C03628=1135.696,-18.528,-48.394,179.412,6.258,149.306
C03629=1135.690,-18.279,-48.406,179.415,6.260,149.305
C03630=1135.685,-18.029,-48.419,179.417,6.261,149.305
C03631=1135.680,-17.780,-48.431,179.420,6.261,149.304
C03632=1135.675,-17.530,-48.443,179.422,6.262,149.304
C03633=1135.669,-17.280,-48.455,179.424,6.263,149.303
C03634=1135.664,-17.031,-48.468,179.427,6.263,149.303
C03635=1135.659,-16.781,-48.480,179.429,6.264,149.302
C03636=1135.654,-16.532,-48.492,179.431,6.265,149.302
C03637=1135.649,-16.282,-48.505,179.434,6.265,149.301
C03638=1135.643,-16.032,-48.517,179.437,6.267,149.300
C03639=1135.639,-15.782,-48.530,179.439,6.267,149.300
C03640=1135.633,-15.533,-48.542,179.442,6.268,149.299
C03641=1135.628,-15.283,-48.554,179.444,6.269,149.299
C03642=1135.623,-15.034,-48.567,179.446,6.269,149.298
C03643=1135.617,-14.784,-48.579,179.449,6.270,149.298
C03644=1135.612,-14.534,-48.592,179.451,6.271,149.297
C03645=1135.607,-14.285,-48.605,179.453,6.271,149.297
C03646=1135.601,-14.036,-48.617,179.456,6.273,149.296
C03647=1135.597,-13.785,-48.629,179.458,6.273,149.296
C03648=1135.591,-13.536,-48.642,179.461,6.274,149.295
C03649=1135.586,-13.286,-48.655,179.463,6.275,149.294
C03650=1135.581,-13.036,-48.667,179.465,6.275,149.294
C03651=1135.576,-12.787,-48.679,179.468,6.276,149.293
C03652=1135.571,-12.538,-48.692,179.470,6.277,149.293
C03653=1135.566,-12.288,-48.705,179.473,6.278,149.292
C03654=1135.561,-12.038,-48.717,179.476,6.279,149.292
C03655=1135.555,-11.788,-48.730,179.478,6.279,149.291
C03656=1135.550,-11.539,-48.742,179.480,6.280,149.291
C03657=1135.545,-11.290,-48.755,179.483,6.281,149.290
C03658=1135.540,-11.039,-48.767,179.485,6.281,149.290
C03659=1135.535,-10.790,-48.780,179.487,6.282,149.289
C03660=1135.529,-10.540,-48.792,179.490,6.283,149.288
C03661=1135.524,-10.291,-48.805,179.493,6.284,149.288
C03662=1135.519,-10.042,-48.818,179.495,6.285,149.287
C03663=1135.514,-9.791,-48.830,179.497,6.285,149.287
C03664=1135.509,-9.541,-48.843,179.500,6.286,149.286
C03665=1135.503,-9.292,-48.856,179.502,6.287,149.286
C03666=1135.498,-9.043,-48.868,179.505,6.288,149.285
C03667=1135.494,-8.793,-48.881,179.507,6.289,149.285
C03668=1135.488,-8.543,-48.894,179.509,6.290,149.284
C03669=1135.483,-8.294,-48.907,179.512,6.290,149.283
C03670=1135.478,-8.045,-48.920,179.514,6.291,149.283
C03671=1135.473,-7.794,-48.932,179.516,6.292,149.283
C03672=1135.468,-7.545,-48.944,179.520,6.293,149.282
C03673=1135.462,-7.295,-48.958,179.522,6.294,149.281
C03674=1135.457,-7.046,-48.970,179.524,6.295,149.281
C03675=1135.452,-6.796,-48.983,179.527,6.295,149.280
C03676=1135.447,-6.546,-48.996,179.529,6.296,149.280
C03677=1135.441,-6.297,-49.009,179.532,6.297,149.279
C03678=1135.436,-6.047,-49.022,179.534,6.298,149.279
C03679=1135.432,-5.797,-49.035,179.536,6.299,149.278
C03680=1135.426,-5.548,-49.047,179.539,6.299,149.277
C03681=1135.421,-5.298,-49.060,179.541,6.300,149.277
C03682=1135.415,-5.049,-49.073,179.544,6.301,149.276
C03683=1135.411,-4.799,-49.086,179.547,6.302,149.276
C03684=1135.405,-4.549,-49.099,179.549,6.303,149.275
C03685=1135.400,-4.300,-49.112,179.551,6.303,149.275
C03686=1135.395,-4.050,-49.125,179.554,6.304,149.274
C03687=1135.390,-3.801,-49.137,179.557,6.305,149.274
C03688=1135.384,-3.551,-49.151,179.559,6.306,149.273
C03689=1135.380,-3.301,-49.163,179.561,6.307,149.273
C03690=1135.375,-3.052,-49.176,179.564,6.307,149.272
C03691=1135.369,-2.802,-49.189,179.566,6.308,149.272
C03692=1135.364,-2.552,-49.202,179.569,6.309,149.271
C03693=1135.359,-2.303,-49.215,179.571,6.310,149.270
C03694=1135.353,-2.053,-49.228,179.573,6.311,149.270
C03695=1135.349,-1.803,-49.241,179.576,6.311,149.269
C03696=1135.343,-1.554,-49.255,179.578,6.312,149.269
C03697=1135.338,-1.305,-49.268,179.581,6.314,149.268
C03698=1135.334,-1.055,-49.280,179.584,6.314,149.268
C03699=1135.328,-0.805,-49.294,179.586,6.315,149.267
C03700=1135.323,-0.556,-49.306,179.588,6.316,149.267
C03701=1135.317,-0.306,-49.320,179.591,6.317,149.266
C03702=1135.312,-0.056,-49.332,179.593,6.318,149.266
C03703=1135.308,0.192,-49.346,179.596,6.319,149.265
C03704=1135.302,0.443,-49.359,179.598,6.319,149.264
C03705=1135.297,0.692,-49.372,179.600,6.320,149.264
C03706=1135.291,0.962,-49.386,179.604,6.321,149.263
C03707=1135.287,1.231,-49.401,179.606,6.322,149.263
C03708=1135.280,1.501,-49.415,179.609,6.323,149.262
C03709=1135.275,1.771,-49.429,179.611,6.324,149.262
C03710=1135.270,2.019,-49.442,179.614,6.324,149.261
C03711=1135.265,2.270,-49.456,179.617,6.326,149.261
C03712=1135.259,2.519,-49.468,179.619,6.327,149.260
C03713=1135.254,2.769,-49.482,179.622,6.327,149.259
C03714=1135.249,3.018,-49.495,179.624,6.328,149.259
C03715=1135.243,3.268,-49.508,179.626,6.330,149.258
C03716=1135.239,3.518,-49.521,179.629,6.330,149.258
C03717=1135.233,3.767,-49.535,179.631,6.331,149.257
C03718=1135.229,4.017,-49.548,179.633,6.332,149.257
C03719=1135.223,4.266,-49.561,179.637,6.333,149.256
C03720=1135.219,4.516,-49.574,179.639,6.334,149.256
C03721=1135.213,4.765,-49.588,179.641,6.334,149.255
C03722=1135.208,5.015,-49.601,179.644,6.335,149.255
C03723=1135.203,5.265,-49.614,179.647,6.336,149.254
C03724=1135.198,5.514,-49.628,179.649,6.337,149.253
C03725=1135.192,5.764,-49.641,179.651,6.338,149.253
C03726=1135.188,6.013,-49.655,179.654,6.339,149.252
C03727=1135.182,6.263,-49.668,179.657,6.340,149.252
C03728=1135.177,6.512,-49.681,179.659,6.341,149.251
C03729=1135.172,6.762,-49.695,179.661,6.341,149.251
C03730=1135.166,7.012,-49.708,179.664,6.342,149.250
C03731=1135.162,7.261,-49.722,179.667,6.343,149.250
C03732=1135.156,7.511,-49.735,179.669,6.344,149.249
C03733=1135.152,7.761,-49.748,179.671,6.345,149.249
C03734=1135.146,8.010,-49.762,179.674,6.346,149.248
C03735=1135.141,8.260,-49.776,179.676,6.347,149.248
C03736=1135.136,8.509,-49.789,179.679,6.347,149.247
C03737=1135.131,8.759,-49.802,179.681,6.348,149.246
C03738=1135.125,9.008,-49.816,179.684,6.350,149.246
C03739=1135.121,9.258,-49.829,179.687,6.350,149.245
C03740=1135.116,9.508,-49.844,179.689,6.351,149.245
C03741=1135.111,9.757,-49.856,179.692,6.353,149.244
C03742=1135.106,10.007,-49.870,179.694,6.353,149.244
C03743=1135.100,10.256,-49.884,179.696,6.354,149.243
C03744=1135.096,10.506,-49.897,179.699,6.356,149.243
C03745=1135.090,10.756,-49.911,179.702,6.356,149.242
C03746=1135.085,11.005,-49.925,179.704,6.357,149.242
C03747=1135.080,11.255,-49.937,179.706,6.358,149.241
C03748=1135.075,11.504,-49.952,179.709,6.359,149.240
C03749=1135.069,11.753,-49.966,179.712,6.360,149.240
C03750=1135.064,12.004,-49.979,179.714,6.360,149.240
C03751=1135.060,12.253,-49.993,179.717,6.362,149.239
C03752=1135.054,12.503,-50.006,179.719,6.362,149.238
C03753=1135.049,12.752,-50.020,179.722,6.363,149.238
C03754=1135.044,13.001,-50.034,179.725,6.364,149.237
C03755=1135.039,13.251,-50.047,179.727,6.365,149.237
C03756=1135.034,13.501,-50.061,179.729,6.366,149.236
C03757=1135.028,13.750,-50.075,179.732,6.367,149.236
C03758=1135.024,14.000,-50.088,179.734,6.368,149.235
C03759=1135.018,14.249,-50.102,179.737,6.369,149.235
C03760=1135.013,14.499,-50.117,179.740,6.370,149.234
C03761=1135.008,14.749,-50.130,179.742,6.371,149.234
C03762=1135.003,14.998,-50.144,179.745,6.371,149.233
C03763=1134.998,15.248,-50.158,179.747,6.373,149.232
C03764=1134.993,15.497,-50.171,179.750,6.374,149.232
C03765=1134.988,15.747,-50.185,179.752,6.374,149.231
C03766=1134.983,15.997,-50.199,179.755,6.376,149.231
C03767=1134.977,16.246,-50.213,179.757,6.377,149.230
C03768=1134.973,16.496,-50.226,179.760,6.377,149.230
C03769=1134.968,16.745,-50.241,179.763,6.379,149.229
C03770=1134.962,16.994,-50.255,179.765,6.380,149.229
C03771=1134.957,17.244,-50.269,179.767,6.380,149.228
C03772=1134.952,17.494,-50.282,179.770,6.382,149.228
C03773=1134.946,17.743,-50.296,179.772,6.382,149.227
C03774=1134.942,17.993,-50.310,179.775,6.383,149.226
C03775=1134.937,18.243,-50.324,179.778,6.384,149.226
C03776=1134.932,18.492,-50.338,179.780,6.385,149.226
C03777=1134.926,18.742,-50.352,179.783,6.386,149.225
C03778=1134.921,18.992,-50.366,179.785,6.387,149.224
C03779=1134.916,19.241,-50.380,179.788,6.388,149.224
C03780=1134.911,19.490,-50.394,179.790,6.389,149.223
C03781=1134.906,19.740,-50.408,179.793,6.390,149.223
C03782=1134.902,19.989,-50.422,179.795,6.391,149.222
C03783=1134.896,20.238,-50.436,179.798,6.391,149.222
C03784=1134.891,20.488,-50.450,179.801,6.393,149.221
C03785=1134.886,20.738,-50.464,179.803,6.394,149.221
C03786=1134.880,20.987,-50.478,179.806,6.395,149.220
C03787=1134.875,21.237,-50.492,179.808,6.396,149.220
C03788=1134.870,21.487,-50.506,179.810,6.397,149.219
C03789=1134.865,21.737,-50.521,179.814,6.398,149.219
C03790=1134.860,21.986,-50.535,179.816,6.399,149.218
C03791=1134.855,22.235,-50.549,179.818,6.400,149.218
C03792=1134.850,22.485,-50.563,179.821,6.401,149.217
C03793=1134.845,22.735,-50.577,179.823,6.402,149.216
C03794=1134.839,22.984,-50.591,179.826,6.403,149.216
C03795=1134.834,23.233,-50.606,179.829,6.404,149.215
C03796=1134.830,23.483,-50.620,179.831,6.404,149.215
C03797=1134.825,23.733,-50.634,179.834,6.406,149.214
C03798=1134.819,23.982,-50.648,179.836,6.407,149.214
C03799=1134.814,24.232,-50.662,179.839,6.408,149.213
C03800=1134.809,24.481,-50.677,179.841,6.409,149.213
C03801=1134.804,24.731,-50.691,179.844,6.409,149.212
C03802=1134.799,24.981,-50.705,179.847,6.411,149.212
C03803=1134.794,25.230,-50.719,179.849,6.412,149.211
C03804=1134.789,25.479,-50.733,179.852,6.413,149.211
C03805=1134.784,25.729,-50.748,179.854,6.414,149.210
C03806=1134.779,25.978,-50.763,179.856,6.415,149.210
C03807=1134.774,26.228,-50.777,179.860,6.416,149.209
C03808=1134.769,26.477,-50.791,179.862,6.417,149.208
C03809=1134.764,26.727,-50.805,179.865,6.418,149.208
C03810=1134.757,26.996,-50.821,179.867,6.419,149.207
C03811=1134.752,27.265,-50.836,179.870,6.420,149.207
C03812=1134.747,27.534,-50.852,179.873,6.421,149.206
C03813=1134.742,27.803,-50.867,179.876,6.422,149.206
C03814=1134.737,28.053,-50.881,179.878,6.423,149.205
C03815=1134.731,28.302,-50.897,179.881,6.425,149.205
C03816=1134.726,28.552,-50.911,179.884,6.425,149.204
C03817=1134.721,28.801,-50.925,179.886,6.427,149.204
C03818=1134.716,29.051,-50.939,179.888,6.427,149.203
C03819=1134.711,29.301,-50.954,179.891,6.429,149.203
C03820=1134.706,29.550,-50.969,179.894,6.429,149.202
C03821=1134.701,29.799,-50.983,179.896,6.430,149.201
C03822=1134.696,30.049,-50.998,179.899,6.432,149.201
C03823=1134.690,30.298,-51.012,179.901,6.432,149.200
C03824=1134.686,30.548,-51.027,179.904,6.434,149.200
C03825=1134.681,30.797,-51.041,179.906,6.435,149.199
C03826=1134.676,31.047,-51.055,179.910,6.436,149.199
C03827=1134.671,31.296,-51.070,179.912,6.437,149.198
C03828=1134.665,31.546,-51.085,179.915,6.439,149.198
C03829=1134.660,31.796,-51.099,179.917,6.439,149.197
C03830=1134.656,32.045,-51.114,179.919,6.440,149.197
C03831=1134.651,32.295,-51.129,179.922,6.441,149.196
C03832=1134.645,32.545,-51.144,179.925,6.442,149.196
C03833=1134.640,32.794,-51.159,179.928,6.443,149.195
C03834=1134.635,33.043,-51.173,179.930,6.444,149.195
C03835=1134.630,33.292,-51.187,179.933,6.446,149.194
C03836=1134.624,33.542,-51.202,179.935,6.446,149.194
C03837=1134.620,33.792,-51.217,179.938,6.448,149.193
C03838=1134.615,34.041,-51.231,179.941,6.448,149.192
C03839=1134.610,34.290,-51.246,179.943,6.450,149.192
C03840=1134.604,34.540,-51.261,179.946,6.451,149.192
C03841=1134.600,34.789,-51.276,179.948,6.451,149.191
C03842=1134.595,35.039,-51.290,179.951,6.453,149.190
C03843=1134.589,35.289,-51.306,179.953,6.454,149.190
C03844=1134.584,35.538,-51.320,179.956,6.455,149.189
C03845=1134.579,35.788,-51.334,179.959,6.456,149.189
C03846=1134.574,36.037,-51.350,179.961,6.457,149.188
C03847=1134.569,36.287,-51.364,179.964,6.458,149.188
C03848=1134.564,36.536,-51.379,179.967,6.460,149.187
C03849=1134.559,36.786,-51.394,179.969,6.460,149.187
C03850=1134.554,37.035,-51.409,179.972,6.462,149.186
C03851=1134.549,37.285,-51.423,179.974,6.462,149.186
C03852=1134.544,37.534,-51.439,179.977,6.464,149.185
C03853=1134.539,37.784,-51.454,179.979,6.465,149.185
C03854=1134.533,38.034,-51.469,179.982,6.466,149.184
C03855=1134.529,38.283,-51.484,179.985,6.467,149.184
C03856=1134.524,38.532,-51.498,179.987,6.469,149.183
C03857=1134.518,38.782,-51.513,179.990,6.469,149.183
C03858=1134.513,39.031,-51.528,179.993,6.471,149.182
C03859=1134.508,39.281,-51.543,179.995,6.471,149.182
C03860=1134.503,39.530,-51.558,179.998,6.473,149.181
C03861=1134.498,39.780,-51.573,-180.000,6.474,149.180
C03862=1134.493,40.029,-51.588,-179.997,6.475,149.180
C03863=1134.488,40.279,-51.602,-179.994,6.476,149.179
C03864=1134.483,40.528,-51.618,-179.991,6.477,149.179
C03865=1134.479,40.778,-51.633,-179.989,6.478,149.178
C03866=1134.473,41.028,-51.648,-179.987,6.480,149.178
C03867=1134.468,41.277,-51.663,-179.984,6.480,149.177
C03868=1134.463,41.526,-51.679,-179.981,6.482,149.177
C03869=1134.458,41.776,-51.693,-179.979,6.483,149.176
C03870=1134.453,42.026,-51.709,-179.976,6.484,149.176
C03871=1134.448,42.275,-51.724,-179.974,6.485,149.175
C03872=1134.442,42.524,-51.739,-179.971,6.486,149.175
C03873=1134.438,42.774,-51.754,-179.968,6.487,149.174
C03874=1134.432,43.023,-51.769,-179.965,6.488,149.174
C03875=1134.428,43.273,-51.785,-179.963,6.489,149.173
C03876=1134.423,43.522,-51.800,-179.960,6.490,149.173
C03877=1134.418,43.772,-51.814,-179.957,6.492,149.172
C03878=1134.412,44.022,-51.830,-179.955,6.493,149.172
C03879=1134.408,44.271,-51.845,-179.952,6.495,149.171
C03880=1134.402,44.520,-51.861,-179.950,6.495,149.171
C03881=1134.398,44.769,-51.876,-179.947,6.497,149.170
C03882=1134.392,45.019,-51.890,-179.945,6.497,149.170
C03883=1134.388,45.269,-51.906,-179.942,6.499,149.169
C03884=1134.383,45.518,-51.921,-179.939,6.500,149.169
C03885=1134.377,45.768,-51.937,-179.937,6.501,149.168
C03886=1134.373,46.017,-51.952,-179.934,6.502,149.167
C03887=1134.367,46.266,-51.968,-179.931,6.503,149.167
C03888=1134.362,46.516,-51.982,-179.928,6.505,149.167
C03889=1134.357,46.766,-51.998,-179.926,6.506,149.166
C03890=1134.352,47.015,-52.013,-179.923,6.507,149.165
C03891=1134.347,47.265,-52.028,-179.921,6.508,149.165
C03892=1134.342,47.514,-52.044,-179.918,6.509,149.165
C03893=1134.337,47.763,-52.060,-179.915,6.510,149.164
C03894=1134.333,48.013,-52.075,-179.913,6.512,149.163
C03895=1134.327,48.263,-52.090,-179.911,6.512,149.163
C03896=1134.322,48.512,-52.105,-179.908,6.514,149.163
C03897=1134.317,48.761,-52.121,-179.905,6.515,149.162
C03898=1134.312,49.010,-52.137,-179.902,6.516,149.161
C03899=1134.308,49.260,-52.152,-179.900,6.518,149.161
C03900=1134.302,49.510,-52.168,-179.897,6.518,149.160
C03901=1134.297,49.759,-52.183,-179.894,6.520,149.160
C03902=1134.292,50.008,-52.199,-179.892,6.521,149.159
C03903=1134.287,50.258,-52.214,-179.889,6.522,149.159
C03904=1134.282,50.508,-52.230,-179.886,6.524,149.158
C03905=1134.277,50.757,-52.245,-179.884,6.524,149.158
C03906=1134.272,51.006,-52.260,-179.881,6.526,149.157
C03907=1134.267,51.256,-52.276,-179.878,6.526,149.157
C03908=1134.262,51.506,-52.292,-179.876,6.528,149.156
C03909=1134.256,51.755,-52.307,-179.873,6.530,149.156
C03910=1134.252,52.005,-52.323,-179.871,6.531,149.155
C03911=1134.247,52.254,-52.338,-179.868,6.532,149.155
C03912=1134.242,52.504,-52.354,-179.865,6.533,149.154
C03913=1134.237,52.752,-52.370,-179.863,6.534,149.154
C03914=1134.231,53.021,-52.387,-179.859,6.536,149.153
C03915=1134.226,53.290,-52.403,-179.857,6.537,149.153
C03916=1134.221,53.559,-52.420,-179.854,6.538,149.152
C03917=1134.215,53.827,-52.437,-179.851,6.539,149.152
C03918=1134.210,54.077,-52.453,-179.848,6.541,149.151
C03919=1134.205,54.327,-52.469,-179.846,6.541,149.151
C03920=1134.200,54.576,-52.485,-179.843,6.543,149.150
C03921=1134.195,54.825,-52.500,-179.840,6.545,149.150
C03922=1134.191,55.075,-52.516,-179.838,6.545,149.149
C03923=1134.185,55.324,-52.532,-179.835,6.547,149.149
C03924=1134.180,55.574,-52.547,-179.833,6.548,149.148
C03925=1134.175,55.823,-52.564,-179.830,6.549,149.148
C03926=1134.170,56.073,-52.580,-179.827,6.550,149.147
C03927=1134.165,56.322,-52.595,-179.825,6.551,149.147
C03928=1134.160,56.572,-52.611,-179.822,6.553,149.146
C03929=1134.156,56.820,-52.627,-179.819,6.555,149.146
C03930=1134.150,57.070,-52.642,-179.816,6.555,149.145
C03931=1134.145,57.320,-52.658,-179.814,6.557,149.145
C03932=1134.140,57.569,-52.675,-179.812,6.557,149.144
C03933=1134.135,57.818,-52.690,-179.808,6.559,149.143
C03934=1134.130,58.068,-52.706,-179.806,6.560,149.143
C03935=1134.125,58.317,-52.723,-179.803,6.561,149.143
C03936=1134.120,58.567,-52.738,-179.801,6.563,149.142
C03937=1134.115,58.817,-52.754,-179.797,6.564,149.142
C03938=1134.110,59.065,-52.770,-179.795,6.565,149.141
C03939=1134.105,59.315,-52.786,-179.793,6.567,149.141
C03940=1134.100,59.564,-52.803,-179.790,6.568,149.140
C03941=1134.095,59.814,-52.819,-179.787,6.569,149.140
C03942=1134.090,60.064,-52.834,-179.784,6.570,149.139
C03943=1134.085,60.313,-52.850,-179.782,6.572,149.139
C03944=1134.080,60.563,-52.866,-179.779,6.573,149.138
C03945=1134.075,60.811,-52.883,-179.776,6.574,149.138
C03946=1134.070,61.062,-52.899,-179.773,6.576,149.137
C03947=1134.065,61.310,-52.915,-179.771,6.577,149.137
C03948=1134.060,61.560,-52.931,-179.769,6.578,149.136
C03949=1134.055,61.809,-52.947,-179.765,6.579,149.136
C03950=1134.050,62.059,-52.963,-179.763,6.580,149.135
C03951=1134.045,62.308,-52.980,-179.760,6.582,149.135
C03952=1134.040,62.558,-52.995,-179.757,6.583,149.134
C03953=1134.035,62.807,-53.012,-179.755,6.584,149.134
C03954=1134.030,63.056,-53.027,-179.752,6.586,149.133
C03955=1134.025,63.306,-53.044,-179.749,6.587,149.133
C03956=1134.020,63.555,-53.060,-179.747,6.588,149.132
C03957=1134.016,63.805,-53.076,-179.744,6.589,149.132
C03958=1134.010,64.054,-53.092,-179.741,6.591,149.131
C03959=1134.006,64.304,-53.109,-179.739,6.592,149.131
C03960=1134.001,64.552,-53.125,-179.736,6.593,149.130
C03961=1133.995,64.803,-53.141,-179.733,6.595,149.130
C03962=1133.991,65.052,-53.158,-179.731,6.596,149.129
C03963=1133.985,65.302,-53.174,-179.728,6.597,149.129
C03964=1133.981,65.551,-53.190,-179.725,6.599,149.128
C03965=1133.976,65.800,-53.207,-179.723,6.599,149.128
C03966=1133.971,66.050,-53.223,-179.720,6.601,149.127
C03967=1133.966,66.299,-53.239,-179.717,6.603,149.127
C03968=1133.961,66.548,-53.256,-179.715,6.604,149.126
C03969=1133.955,66.798,-53.272,-179.712,6.605,149.126
C03970=1133.951,67.048,-53.288,-179.709,6.607,149.125
C03971=1133.946,67.296,-53.305,-179.707,6.608,149.125
C03972=1133.941,67.546,-53.321,-179.704,6.609,149.124
C03973=1133.936,67.796,-53.337,-179.701,6.610,149.124
C03974=1133.931,68.045,-53.354,-179.698,6.612,149.123
C03975=1133.926,68.294,-53.371,-179.696,6.614,149.123
C03976=1133.921,68.544,-53.386,-179.693,6.614,149.122
C03977=1133.916,68.793,-53.403,-179.690,6.616,149.122
C03978=1133.911,69.042,-53.419,-179.687,6.617,149.121
C03979=1133.906,69.292,-53.437,-179.685,6.618,149.121
C03980=1133.901,69.541,-53.453,-179.683,6.620,149.120
C03981=1133.896,69.791,-53.469,-179.679,6.621,149.120
C03982=1133.892,70.040,-53.486,-179.677,6.623,149.119
C03983=1133.886,70.289,-53.503,-179.674,6.624,149.119
C03984=1133.881,70.539,-53.519,-179.672,6.625,149.118
C03985=1133.877,70.788,-53.536,-179.669,6.627,149.118
C03986=1133.871,71.037,-53.553,-179.666,6.628,149.117
C03987=1133.866,71.288,-53.569,-179.664,6.629,149.117
C03988=1133.862,71.537,-53.585,-179.661,6.631,149.117
C03989=1133.857,71.786,-53.602,-179.658,6.632,149.116
C03990=1133.851,72.036,-53.619,-179.655,6.633,149.115
C03991=1133.846,72.284,-53.635,-179.653,6.634,149.115
C03992=1133.842,72.534,-53.652,-179.650,6.636,149.115
C03993=1133.837,72.784,-53.669,-179.647,6.638,149.114
C03994=1133.832,73.032,-53.686,-179.645,6.639,149.114
C03995=1133.827,73.282,-53.702,-179.642,6.640,149.113
C03996=1133.822,73.532,-53.719,-179.639,6.641,149.113
C03997=1133.817,73.781,-53.736,-179.636,6.643,149.112
C03998=1133.812,74.030,-53.753,-179.634,6.645,149.112
C03999=1133.807,74.280,-53.770,-179.631,6.645,149.111
C04000=1133.803,74.529,-53.786,-179.628,6.647,149.111
C04001=1133.797,74.778,-53.803,-179.625,6.649,149.110
C04002=1133.792,75.028,-53.820,-179.623,6.650,149.110
C04003=1133.787,75.278,-53.837,-179.621,6.651,149.109
C04004=1133.782,75.526,-53.853,-179.617,6.652,149.109
C04005=1133.778,75.776,-53.870,-179.615,6.654,149.108
C04006=1133.772,76.026,-53.887,-179.612,6.656,149.108
C04007=1133.768,76.275,-53.904,-179.610,6.656,149.107
C04008=1133.762,76.524,-53.921,-179.607,6.658,149.107
C04009=1133.758,76.774,-53.938,-179.604,6.659,149.106
C04010=1133.752,77.024,-53.955,-179.601,6.661,149.106
C04011=1133.747,77.272,-53.971,-179.598,6.663,149.105
C04012=1133.742,77.522,-53.989,-179.596,6.664,149.105
C04013=1133.738,77.771,-54.006,-179.593,6.665,149.105
C04014=1133.733,78.021,-54.023,-179.590,6.667,149.104
C04015=1133.728,78.270,-54.039,-179.587,6.668,149.104
C04016=1133.722,78.519,-54.057,-179.585,6.669,149.103
C04017=1133.718,78.769,-54.073,-179.582,6.671,149.103
C04018=1133.712,79.038,-54.092,-179.579,6.672,149.102
C04019=1133.707,79.306,-54.110,-179.576,6.674,149.102
C04020=1133.702,79.575,-54.129,-179.574,6.675,149.101
C04021=1133.697,79.842,-54.147,-179.570,6.677,149.101
C04022=1133.692,80.092,-54.164,-179.568,6.678,149.100
C04023=1133.686,80.341,-54.181,-179.565,6.680,149.100
C04024=1133.682,80.591,-54.198,-179.562,6.681,149.099
C04025=1133.677,80.840,-54.216,-179.559,6.683,149.099
C04026=1133.672,81.089,-54.232,-179.557,6.684,149.098
C04027=1133.667,81.339,-54.250,-179.554,6.685,149.098
C04028=1133.662,81.588,-54.266,-179.551,6.687,149.097
C04029=1133.657,81.837,-54.284,-179.549,6.689,149.097
C04030=1133.652,82.087,-54.302,-179.546,6.690,149.096
C04031=1133.648,82.337,-54.318,-179.543,6.691,149.096
C04032=1133.642,82.585,-54.336,-179.540,6.692,149.095
C04033=1133.637,82.835,-54.353,-179.538,6.694,149.095
C04034=1133.632,83.084,-54.370,-179.535,6.696,149.095
C04035=1133.628,83.333,-54.388,-179.532,6.697,149.094
C04036=1133.623,83.583,-54.404,-179.529,6.699,149.093
C04037=1133.618,83.832,-54.422,-179.527,6.699,149.093
C04038=1133.613,84.082,-54.440,-179.524,6.701,149.093
C04039=1133.608,84.331,-54.456,-179.521,6.703,149.092
C04040=1133.603,84.580,-54.474,-179.519,6.704,149.092
C04041=1133.598,84.830,-54.491,-179.516,6.706,149.091
C04042=1133.594,85.079,-54.509,-179.513,6.707,149.091
C04043=1133.588,85.328,-54.526,-179.510,6.708,149.090
C04044=1133.583,85.577,-54.544,-179.508,6.710,149.090
C04045=1133.578,85.827,-54.561,-179.505,6.712,149.089
C04046=1133.574,86.076,-54.579,-179.502,6.713,149.089
C04047=1133.569,86.326,-54.596,-179.500,6.715,149.089
C04048=1133.564,86.575,-54.614,-179.496,6.716,149.088
C04049=1133.559,86.825,-54.631,-179.494,6.718,149.087
C04050=1133.554,87.073,-54.648,-179.491,6.719,149.087
C04051=1133.549,87.323,-54.665,-179.489,6.720,149.087
C04052=1133.544,87.572,-54.683,-179.486,6.722,149.086
C04053=1133.539,87.822,-54.701,-179.483,6.724,149.086
C04054=1133.534,88.071,-54.718,-179.480,6.725,149.085
C04055=1133.529,88.320,-54.736,-179.477,6.727,149.085
C04056=1133.524,88.570,-54.753,-179.474,6.728,149.084
C04057=1133.519,88.819,-54.771,-179.472,6.730,149.084
C04058=1133.514,89.069,-54.788,-179.470,6.731,149.083
C04059=1133.510,89.318,-54.806,-179.467,6.732,149.083
C04060=1133.505,89.567,-54.824,-179.464,6.734,149.082
C04061=1133.500,89.816,-54.841,-179.461,6.735,149.082
C04062=1133.495,90.066,-54.859,-179.458,6.737,149.082
C04063=1133.490,90.315,-54.877,-179.455,6.739,149.081
C04064=1133.485,90.565,-54.894,-179.453,6.740,149.081
C04065=1133.481,90.813,-54.912,-179.450,6.742,149.080
C04066=1133.476,91.063,-54.930,-179.448,6.743,149.080
C04067=1133.470,91.312,-54.947,-179.445,6.744,149.079
C04068=1133.466,91.562,-54.965,-179.442,6.746,149.079
C04069=1133.461,91.811,-54.983,-179.439,6.748,149.078
C04070=1133.456,92.060,-55.001,-179.436,6.749,149.078
C04071=1133.450,92.310,-55.018,-179.434,6.751,149.077
C04072=1133.446,92.559,-55.036,-179.431,6.753,149.077
C04073=1133.441,92.808,-55.054,-179.428,6.754,149.077
C04074=1133.436,93.057,-55.071,-179.425,6.755,149.076
C04075=1133.431,93.307,-55.089,-179.422,6.757,149.076
C04076=1133.426,93.556,-55.107,-179.420,6.758,149.075
C04077=1133.421,93.805,-55.125,-179.417,6.760,149.075
C04078=1133.417,94.054,-55.143,-179.414,6.761,149.074
C04079=1133.412,94.304,-55.161,-179.412,6.763,149.074
C04080=1133.407,94.553,-55.179,-179.409,6.765,149.073
C04081=1133.402,94.803,-55.196,-179.406,6.766,149.073
C04082=1133.397,95.052,-55.214,-179.403,6.768,149.072
C04083=1133.392,95.302,-55.232,-179.400,6.769,149.072
C04084=1133.387,95.551,-55.250,-179.398,6.771,149.072
C04085=1133.382,95.800,-55.268,-179.395,6.773,149.071
C04086=1133.378,96.049,-55.286,-179.392,6.774,149.071
C04087=1133.373,96.298,-55.304,-179.389,6.776,149.070
C04088=1133.368,96.547,-55.322,-179.387,6.778,149.070
C04089=1133.363,96.797,-55.340,-179.384,6.778,149.069
C04090=1133.358,97.046,-55.358,-179.381,6.780,149.069
C04091=1133.354,97.296,-55.376,-179.378,6.781,149.068
C04092=1133.349,97.545,-55.394,-179.376,6.783,149.068
C04093=1133.343,97.794,-55.413,-179.373,6.785,149.068
C04094=1133.338,98.043,-55.431,-179.370,6.786,149.067
C04095=1133.333,98.293,-55.449,-179.368,6.788,149.067
C04096=1133.328,98.542,-55.467,-179.365,6.790,149.066
C04097=1133.324,98.792,-55.485,-179.362,6.791,149.066
C04098=1133.319,99.041,-55.503,-179.359,6.793,149.065
C04099=1133.314,99.290,-55.521,-179.356,6.794,149.065
C04100=1133.309,99.539,-55.539,-179.353,6.796,149.064
C04101=1133.304,99.788,-55.557,-179.351,6.798,149.064
C04102=1133.300,100.038,-55.576,-179.348,6.799,149.064
C04103=1133.294,100.288,-55.594,-179.345,6.801,149.063
C04104=1133.289,100.537,-55.612,-179.342,6.803,149.063
C04105=1133.285,100.786,-55.630,-179.340,6.804,149.062
C04106=1133.280,101.035,-55.649,-179.337,6.806,149.062
C04107=1133.276,101.285,-55.667,-179.334,6.808,149.062
C04108=1133.271,101.534,-55.685,-179.331,6.809,149.061
C04109=1133.265,101.783,-55.704,-179.328,6.811,149.060
C04110=1133.260,102.032,-55.722,-179.325,6.812,149.060
C04111=1133.255,102.282,-55.740,-179.323,6.814,149.060
C04112=1133.251,102.531,-55.759,-179.320,6.816,149.059
C04113=1133.246,102.780,-55.777,-179.318,6.817,149.059
C04114=1133.241,103.029,-55.795,-179.315,6.818,149.058
C04115=1133.236,103.279,-55.813,-179.312,6.820,149.058
C04116=1133.232,103.528,-55.832,-179.310,6.822,149.058
C04117=1133.227,103.777,-55.850,-179.307,6.823,149.057
C04118=1133.221,104.027,-55.869,-179.304,6.825,149.057
C04119=1133.216,104.276,-55.887,-179.301,6.826,149.056
C04120=1133.212,104.525,-55.906,-179.298,6.828,149.056
C04121=1133.207,104.774,-55.924,-179.295,6.830,149.055
C04122=1133.202,105.043,-55.944,-179.292,6.832,149.055
C04123=1133.196,105.311,-55.963,-179.289,6.834,149.054
C04124=1133.191,105.579,-55.984,-179.287,6.835,149.054
C04125=1133.186,105.848,-56.004,-179.283,6.837,149.053
C04126=1133.181,106.097,-56.022,-179.281,6.838,149.053
C04127=1133.176,106.346,-56.041,-179.278,6.840,149.053
C04128=1133.172,106.596,-56.059,-179.275,6.842,149.052
C04129=1133.166,106.845,-56.078,-179.273,6.843,149.052
C04130=1133.162,107.094,-56.097,-179.270,6.845,149.051
C04131=1133.157,107.344,-56.115,-179.267,6.847,149.051
C04132=1133.152,107.593,-56.134,-179.264,6.848,149.051
C04133=1133.147,107.842,-56.152,-179.262,6.850,149.050
C04134=1133.143,108.092,-56.171,-179.259,6.852,149.050
C04135=1133.137,108.341,-56.190,-179.256,6.853,149.049
C04136=1133.133,108.590,-56.208,-179.253,6.856,149.049
C04137=1133.128,108.839,-56.228,-179.250,6.858,149.048
C04138=1133.123,109.088,-56.246,-179.247,6.859,149.048
C04139=1133.118,109.337,-56.264,-179.244,6.861,149.047
C04140=1133.113,109.587,-56.283,-179.241,6.862,149.047
C04141=1133.109,109.836,-56.302,-179.239,6.864,149.047
C04142=1133.104,110.086,-56.321,-179.236,6.866,149.046
C04143=1133.099,110.334,-56.339,-179.233,6.867,149.046
C04144=1133.094,110.583,-56.359,-179.230,6.869,149.045
C04145=1133.089,110.833,-56.377,-179.228,6.871,149.045
C04146=1133.084,111.082,-56.396,-179.225,6.872,149.045
C04147=1133.079,111.331,-56.414,-179.222,6.874,149.044
C04148=1133.074,111.581,-56.434,-179.219,6.876,149.044
C04149=1133.070,111.829,-56.453,-179.217,6.877,149.043
C04150=1133.065,112.080,-56.472,-179.214,6.879,149.043
C04151=1133.060,112.328,-56.490,-179.211,6.881,149.043
C04152=1133.055,112.578,-56.509,-179.209,6.882,149.042
C04153=1133.050,112.827,-56.528,-179.206,6.884,149.042
C04154=1133.045,113.076,-56.547,-179.203,6.886,149.041
C04155=1133.041,113.326,-56.566,-179.200,6.887,149.041
C04156=1133.035,113.575,-56.585,-179.198,6.889,149.040
C04157=1133.031,113.824,-56.604,-179.194,6.891,149.040
C04158=1133.026,114.073,-56.623,-179.192,6.893,149.040
C04159=1133.021,114.323,-56.642,-179.189,6.895,149.039
C04160=1133.016,114.571,-56.661,-179.186,6.896,149.039
C04161=1133.012,114.821,-56.681,-179.183,6.898,149.038
C04162=1133.007,115.070,-56.699,-179.181,6.900,149.038
C04163=1133.002,115.320,-56.718,-179.178,6.902,149.038
C04164=1132.997,115.569,-56.738,-179.175,6.903,149.037
C04165=1132.993,115.818,-56.757,-179.172,6.905,149.037
C04166=1132.987,116.067,-56.776,-179.169,6.906,149.036
C04167=1132.983,116.317,-56.794,-179.166,6.908,149.036
C04168=1132.978,116.565,-56.814,-179.164,6.910,149.035
C04169=1132.973,116.815,-56.833,-179.160,6.912,149.035
C04170=1132.968,117.064,-56.852,-179.158,6.914,149.035
C04171=1132.964,117.313,-56.872,-179.155,6.915,149.034
C04172=1132.958,117.562,-56.891,-179.152,6.917,149.034
C04173=1132.954,117.811,-56.910,-179.150,6.919,149.033
C04174=1132.949,118.061,-56.928,-179.147,6.920,149.033
C04175=1132.944,118.310,-56.948,-179.144,6.922,149.033
C04176=1132.939,118.559,-56.967,-179.141,6.924,149.032
C04177=1132.934,118.808,-56.986,-179.139,6.925,149.032
C04178=1132.929,119.057,-57.006,-179.136,6.927,149.031
C04179=1132.924,119.307,-57.025,-179.133,6.930,149.031
C04180=1132.920,119.556,-57.044,-179.130,6.931,149.031
C04181=1132.915,119.805,-57.064,-179.127,6.933,149.030
C04182=1132.910,120.055,-57.083,-179.124,6.935,149.030
C04183=1132.905,120.303,-57.103,-179.122,6.936,149.029
C04184=1132.901,120.553,-57.122,-179.119,6.938,149.029
C04185=1132.896,120.802,-57.141,-179.116,6.940,149.029
C04186=1132.891,121.051,-57.161,-179.113,6.941,149.028
C04187=1132.886,121.301,-57.180,-179.110,6.944,149.028
C04188=1132.881,121.549,-57.199,-179.107,6.946,149.027
C04189=1132.877,121.799,-57.219,-179.105,6.947,149.027
C04190=1132.872,122.048,-57.238,-179.102,6.949,149.027
C04191=1132.867,122.297,-57.258,-179.100,6.951,149.026
C04192=1132.862,122.546,-57.278,-179.097,6.953,149.026
C04193=1132.857,122.795,-57.297,-179.094,6.954,149.026
C04194=1132.853,123.044,-57.316,-179.091,6.957,149.025
C04195=1132.848,123.294,-57.336,-179.088,6.959,149.025
C04196=1132.843,123.543,-57.355,-179.085,6.960,149.024
C04197=1132.838,123.792,-57.375,-179.083,6.962,149.024
C04198=1132.833,124.042,-57.395,-179.080,6.964,149.024
C04199=1132.828,124.290,-57.415,-179.077,6.965,149.023
C04200=1132.823,124.540,-57.434,-179.074,6.967,149.023
C04201=1132.819,124.789,-57.453,-179.071,6.969,149.022
C04202=1132.814,125.038,-57.473,-179.068,6.971,149.022
C04203=1132.809,125.287,-57.492,-179.066,6.973,149.022
C04204=1132.805,125.536,-57.513,-179.063,6.974,149.021
C04205=1132.800,125.786,-57.532,-179.060,6.976,149.021
C04206=1132.795,126.035,-57.552,-179.058,6.978,149.020
C04207=1132.790,126.284,-57.571,-179.054,6.980,149.020
C04208=1132.786,126.533,-57.592,-179.051,6.982,149.020
C04209=1132.780,126.782,-57.611,-179.049,6.984,149.019
C04210=1132.776,127.032,-57.631,-179.046,6.985,149.019
C04211=1132.771,127.281,-57.651,-179.043,6.987,149.018
C04212=1132.766,127.530,-57.671,-179.041,6.989,149.018
C04213=1132.761,127.779,-57.690,-179.037,6.991,149.018
C04214=1132.757,128.028,-57.710,-179.035,6.993,149.017
C04215=1132.752,128.278,-57.730,-179.032,6.995,149.017
C04216=1132.747,128.527,-57.750,-179.030,6.997,149.017
C04217=1132.742,128.775,-57.770,-179.027,6.998,149.016
C04218=1132.737,129.025,-57.789,-179.024,7.001,149.016
C04219=1132.733,129.274,-57.810,-179.021,7.003,149.015
C04220=1132.728,129.524,-57.829,-179.018,7.004,149.015
C04221=1132.723,129.772,-57.849,-179.015,7.006,149.015
C04222=1132.718,130.021,-57.869,-179.013,7.008,149.014
C04223=1132.714,130.271,-57.889,-179.009,7.010,149.014
C04224=1132.709,130.520,-57.909,-179.007,7.012,149.013
C04225=1132.705,130.769,-57.929,-179.004,7.013,149.013
C04226=1132.699,131.038,-57.951,-179.001,7.015,149.013
C04227=1132.694,131.306,-57.972,-178.998,7.018,149.012
C04228=1132.688,131.575,-57.993,-178.995,7.019,149.012
C04229=1132.683,131.843,-58.015,-178.992,7.022,149.011
C04230=1132.679,132.092,-58.035,-178.989,7.023,149.011
C04231=1132.674,132.341,-58.055,-178.986,7.025,149.011
C04232=1132.669,132.591,-58.075,-178.984,7.027,149.010
C04233=1132.664,132.840,-58.096,-178.980,7.029,149.010
C04234=1132.660,133.090,-58.116,-178.978,7.031,149.010
C04235=1132.655,133.338,-58.136,-178.975,7.033,149.009
C04236=1132.650,133.587,-58.156,-178.972,7.034,149.009
C04237=1132.645,133.836,-58.176,-178.969,7.037,149.009
C04238=1132.641,134.085,-58.196,-178.967,7.039,149.008
C04239=1132.636,134.335,-58.217,-178.964,7.041,149.008
C04240=1132.631,134.584,-58.237,-178.961,7.042,149.007
C04241=1132.627,134.833,-58.257,-178.958,7.044,149.007
C04242=1132.622,135.082,-58.277,-178.955,7.047,149.007
C04243=1132.616,135.331,-58.297,-178.952,7.048,149.006
C04244=1132.612,135.580,-58.318,-178.950,7.050,149.006
C04245=1132.607,135.829,-58.338,-178.947,7.052,149.005
C04246=1132.602,136.079,-58.358,-178.944,7.054,149.005
C04247=1132.597,136.328,-58.379,-178.941,7.056,149.005
C04248=1132.593,136.577,-58.399,-178.939,7.058,149.004
C04249=1132.588,136.826,-58.419,-178.936,7.060,149.004
C04250=1132.584,137.075,-58.439,-178.933,7.062,149.004
C04251=1132.578,137.325,-58.460,-178.930,7.064,149.003
C04252=1132.574,137.574,-58.480,-178.927,7.065,149.003
C04253=1132.570,137.823,-58.501,-178.924,7.067,149.003
C04254=1132.564,138.072,-58.522,-178.921,7.070,149.002
C04255=1132.560,138.321,-58.542,-178.918,7.071,149.002
C04256=1132.555,138.570,-58.561,-178.916,7.073,149.002
C04257=1132.549,138.819,-58.582,-178.913,7.076,149.001
C04258=1132.530,139.892,-58.674,-179.676,8.531,149.554
C04259=1132.525,140.141,-58.694,-179.675,8.535,149.554
C04260=1132.520,140.391,-58.715,-179.673,8.538,149.554
C04261=1132.516,140.640,-58.736,-179.672,8.541,149.555
C04262=1132.511,140.889,-58.757,-179.670,8.545,149.555
C04263=1132.506,141.138,-58.777,-179.669,8.548,149.555
C04264=1132.501,141.386,-58.799,-179.668,8.551,149.556
C04265=1132.497,141.635,-58.819,-179.666,8.554,149.556
C04266=1132.492,141.885,-58.840,-179.665,8.557,149.557
C04267=1132.488,142.134,-58.861,-179.662,8.561,149.557
C04268=1132.483,142.384,-58.882,-179.661,8.564,149.557
C04269=1132.478,142.633,-58.902,-179.660,8.567,149.558
C04270=1132.473,142.881,-58.924,-179.658,8.571,149.558
C04271=1132.468,143.130,-58.945,-179.657,8.574,149.558
C04272=1132.464,143.379,-58.965,-179.656,8.577,149.559
C04273=1132.459,143.629,-58.986,-179.654,8.580,149.559
C04274=1132.455,143.878,-59.008,-179.653,8.583,149.559
C04275=1132.449,144.159,-59.031,-179.652,8.587,149.560
C04276=1132.444,144.440,-59.055,-179.650,8.591,149.560
C04277=1132.439,144.722,-59.079,-179.648,8.595,149.561
C04278=1132.433,145.004,-59.102,-179.647,8.599,149.561
C04279=1132.428,145.253,-59.124,-179.644,8.603,149.561
C04280=1132.424,145.501,-59.144,-179.641,8.607,149.561
C04281=1132.419,145.751,-59.165,-179.639,8.610,149.562
C04282=1132.414,146.000,-59.187,-179.636,8.615,149.562
C04283=1132.410,146.249,-59.207,-179.633,8.619,149.562
C04284=1132.405,146.498,-59.229,-179.630,8.623,149.562
C04285=1132.400,146.747,-59.250,-179.627,8.627,149.562
C04286=1132.395,146.996,-59.270,-179.624,8.631,149.562
C04287=1132.391,147.245,-59.292,-179.622,8.635,149.563
C04288=1132.386,147.494,-59.313,-179.618,8.639,149.563
C04289=1132.381,147.743,-59.335,-179.616,8.643,149.563
C04290=1132.377,147.992,-59.355,-179.613,8.646,149.563
C04291=1132.372,148.241,-59.378,-179.611,8.651,149.563
C04292=1132.367,148.491,-59.398,-179.607,8.655,149.563
C04293=1132.362,148.739,-59.420,-179.605,8.659,149.563
C04294=1132.358,148.988,-59.441,-179.602,8.663,149.564
C04295=1132.354,149.238,-59.463,-179.599,8.666,149.564
C04296=1132.348,149.487,-59.484,-179.597,8.671,149.564
C04297=1132.344,149.736,-59.505,-179.594,8.674,149.564
C04298=1132.339,149.984,-59.527,-179.591,8.679,149.564
C04299=1132.334,150.234,-59.548,-179.588,8.682,149.564
C04300=1132.330,150.482,-59.569,-179.586,8.686,149.564
C04301=1132.325,150.732,-59.590,-179.582,8.690,149.564
C04302=1132.321,150.981,-59.612,-179.580,8.693,149.564
C04303=1132.316,151.230,-59.634,-179.577,8.697,149.565
C04304=1132.311,151.479,-59.655,-179.574,8.701,149.565
C04305=1132.306,151.728,-59.677,-179.572,8.705,149.565
C04306=1132.301,151.977,-59.699,-179.569,8.709,149.565
C04307=1132.296,152.226,-59.720,-179.566,8.713,149.565
C04308=1132.292,152.476,-59.742,-179.564,8.716,149.565
C04309=1132.287,152.724,-59.763,-179.561,8.720,149.565
C04310=1132.282,152.973,-59.785,-179.558,8.723,149.565
C04311=1132.278,153.222,-59.807,-179.555,8.727,149.565
C04312=1132.273,153.471,-59.828,-179.553,8.731,149.566
C04313=1132.269,153.720,-59.849,-179.550,8.735,149.566
C04314=1132.264,153.969,-59.871,-179.547,8.739,149.566
C04315=1132.259,154.218,-59.893,-179.545,8.742,149.566
C04316=1132.255,154.467,-59.915,-179.542,8.746,149.566
C04317=1132.250,154.716,-59.937,-179.539,8.749,149.566
C04318=1132.245,154.965,-59.959,-179.536,8.753,149.566
C04319=1132.240,155.215,-59.980,-179.534,8.756,149.566
C04320=1132.235,155.463,-60.002,-179.531,8.761,149.567
C04321=1132.231,155.713,-60.024,-179.529,8.764,149.567
C04322=1132.226,155.961,-60.046,-179.526,8.767,149.567
C04323=1132.222,156.211,-60.068,-179.523,8.771,149.567
C04324=1132.217,156.459,-60.089,-179.521,8.774,149.567
C04325=1132.212,156.708,-60.111,-179.518,8.778,149.567
C04326=1132.208,156.957,-60.133,-179.516,8.781,149.567
C04327=1132.204,157.171,-60.152,-179.513,8.785,149.567
C04328=1132.200,157.387,-60.171,-179.511,8.788,149.567
C04329=1132.196,157.601,-60.190,-179.509,8.790,149.567
C04330=1132.192,157.816,-60.208,-179.507,8.794,149.567
C04331=1132.188,158.031,-60.228,-179.504,8.797,149.567
C04332=1132.184,158.245,-60.247,-179.501,8.800,149.567
C04333=1132.180,158.460,-60.265,-179.500,8.802,149.568
C04334=1132.176,158.675,-60.285,-179.498,8.806,149.568
C04335=1132.170,158.924,-60.307,-179.495,8.809,149.568
C04336=1132.166,159.173,-60.329,-179.492,8.813,149.568
C04337=1132.161,159.422,-60.351,-179.489,8.816,149.568
C04338=1132.157,159.670,-60.374,-179.487,8.819,149.568
C04339=1132.153,159.919,-60.395,-179.484,8.823,149.568
C04340=1132.147,160.169,-60.418,-179.482,8.826,149.568
C04341=1132.143,160.417,-60.440,-179.479,8.830,149.568
C04342=1132.138,160.667,-60.462,-179.477,8.833,149.568
C04343=1132.134,160.916,-60.484,-179.474,8.837,149.568
C04344=1132.130,161.164,-60.506,-179.471,8.840,149.568
C04345=1132.125,161.414,-60.529,-179.469,8.843,149.569
C04346=1132.120,161.662,-60.550,-179.467,8.846,149.569
C04347=1132.116,161.911,-60.573,-179.464,8.849,149.569
C04348=1132.110,162.160,-60.595,-179.461,8.853,149.569
C04349=1132.106,162.409,-60.618,-179.458,8.856,149.569
C04350=1132.102,162.659,-60.640,-179.456,8.860,149.569
C04351=1132.097,162.907,-60.662,-179.454,8.863,149.569
C04352=1132.092,163.156,-60.685,-179.451,8.866,149.569
C04353=1132.087,163.405,-60.706,-179.449,8.869,149.569
C04354=1132.083,163.654,-60.729,-179.447,8.873,149.569
C04355=1132.078,163.903,-60.752,-179.444,8.876,149.569
C04356=1132.074,164.151,-60.774,-179.441,8.880,149.569
C04357=1132.069,164.401,-60.796,-179.439,8.883,149.569
C04358=1132.064,164.650,-60.819,-179.436,8.886,149.570
C04359=1132.060,164.898,-60.841,-179.434,8.889,149.570
C04360=1132.055,165.148,-60.864,-179.431,8.892,149.570
C04361=1132.051,165.397,-60.887,-179.429,8.896,149.570
C04362=1132.046,165.645,-60.908,-179.426,8.899,149.570
C04363=1132.041,165.894,-60.932,-179.424,8.902,149.570
C04364=1132.037,166.144,-60.954,-179.422,8.905,149.570
C04365=1132.032,166.392,-60.977,-179.419,8.908,149.570
C04366=1132.027,166.641,-60.999,-179.417,8.912,149.570
C04367=1132.023,166.890,-61.022,-179.414,8.915,149.570
C04368=1132.018,167.139,-61.044,-179.412,8.918,149.570
C04369=1132.013,167.388,-61.067,-179.410,8.921,149.570
C04370=1132.009,167.637,-61.089,-179.407,8.924,149.571
C04371=1132.004,167.886,-61.112,-179.404,8.927,149.571
C04372=1132.000,168.135,-61.135,-179.402,8.931,149.571
C04373=1131.995,168.384,-61.158,-179.400,8.934,149.571
C04374=1131.991,168.633,-61.180,-179.397,8.937,149.571
C04375=1131.985,168.881,-61.203,-179.395,8.939,149.571
C04376=1131.981,169.131,-61.225,-179.393,8.943,149.571
C04377=1131.976,169.380,-61.249,-179.391,8.946,149.571
C04378=1131.972,169.628,-61.271,-179.388,8.949,149.571
C04379=1131.967,169.877,-61.294,-179.386,8.952,149.571
C04380=1131.963,170.126,-61.317,-179.383,8.955,149.571
C04381=1131.958,170.375,-61.340,-179.381,8.959,149.571
C04382=1131.953,170.625,-61.363,-179.379,8.962,149.572
C04383=1131.949,170.838,-61.382,-179.377,8.964,149.572
C04384=1131.946,171.053,-61.402,-179.375,8.967,149.572
C04385=1131.941,171.268,-61.421,-179.373,8.969,149.572
C04386=1131.938,171.483,-61.441,-179.371,8.972,149.572
C04387=1131.933,171.698,-61.461,-179.369,8.975,149.572
C04388=1131.930,171.911,-61.481,-179.367,8.977,149.572
C04389=1131.925,172.127,-61.501,-179.365,8.980,149.572
C04390=1131.921,172.341,-61.520,-179.363,8.983,149.572
C04391=1131.917,172.590,-61.543,-179.361,8.986,149.572
C04392=1131.913,172.838,-61.566,-179.359,8.988,149.572
C04393=1131.908,173.088,-61.589,-179.356,8.991,149.572
C04394=1131.903,173.337,-61.613,-179.354,8.995,149.572
C04395=1131.899,173.585,-61.635,-179.352,8.998,149.573
C04396=1131.894,173.834,-61.658,-179.350,9.000,149.573
C04397=1131.889,174.083,-61.681,-179.347,9.003,149.573
C04398=1131.885,174.332,-61.704,-179.345,9.007,149.573
C04399=1131.880,174.581,-61.727,-179.342,9.010,149.573
C04400=1131.876,174.830,-61.751,-179.341,9.012,149.573
C04401=1131.871,175.079,-61.774,-179.339,9.016,149.573
C04402=1131.866,175.327,-61.796,-179.336,9.019,149.573
C04403=1131.862,175.576,-61.820,-179.334,9.021,149.573
C04404=1131.857,175.825,-61.843,-179.332,9.025,149.573
C04405=1131.852,176.074,-61.866,-179.329,9.028,149.573
C04406=1131.848,176.323,-61.889,-179.328,9.030,149.574
C04407=1131.844,176.572,-61.913,-179.325,9.033,149.574
C04408=1131.839,176.821,-61.936,-179.323,9.037,149.574
C04409=1131.834,177.070,-61.959,-179.321,9.039,149.574
C04410=1131.830,177.319,-61.982,-179.319,9.042,149.574
C04411=1131.825,177.567,-62.005,-179.317,9.045,149.574
C04412=1131.820,177.816,-62.028,-179.315,9.048,149.574
C04413=1131.815,178.065,-62.052,-179.312,9.052,149.574
C04414=1131.811,178.314,-62.075,-179.311,9.054,149.574
C04415=1131.806,178.563,-62.099,-179.308,9.057,149.574
C04416=1131.802,178.811,-62.122,-179.307,9.060,149.575
C04417=1131.798,179.060,-62.145,-179.304,9.063,149.575
C04418=1131.793,179.309,-62.169,-179.302,9.066,149.575
C04419=1131.788,179.558,-62.192,-179.298,9.070,149.575
C04420=1131.784,179.807,-62.215,-179.295,9.073,149.575
C04421=1131.779,180.056,-62.239,-179.292,9.076,149.575
C04422=1131.774,180.305,-62.262,-179.289,9.080,149.575
C04423=1131.771,180.554,-62.286,-179.286,9.084,149.575
C04424=1131.766,180.803,-62.309,-179.283,9.087,149.575
C04425=1131.761,181.052,-62.332,-179.279,9.090,149.574
C04426=1131.756,181.301,-62.356,-179.277,9.093,149.574
C04427=1131.752,181.549,-62.380,-179.273,9.097,149.574
C04428=1131.747,181.798,-62.403,-179.271,9.100,149.574
C04429=1131.743,182.047,-62.426,-179.268,9.104,149.574
C04430=1131.738,182.296,-62.451,-179.265,9.107,149.574
C04431=1131.734,182.545,-62.474,-179.261,9.111,149.574
C04432=1131.729,182.794,-62.497,-179.259,9.114,149.574
C04433=1131.724,183.042,-62.521,-179.256,9.116,149.574
C04434=1131.720,183.291,-62.545,-179.253,9.120,149.574
C04435=1131.715,183.540,-62.568,-179.250,9.123,149.574
C04436=1131.711,183.789,-62.592,-179.247,9.126,149.574
C04437=1131.706,184.038,-62.616,-179.245,9.129,149.574
C04438=1131.702,184.286,-62.640,-179.242,9.132,149.574
C04439=1131.698,184.501,-62.660,-179.240,9.135,149.574
C04440=1131.693,184.716,-62.680,-179.237,9.137,149.574
C04441=1131.690,184.930,-62.701,-179.235,9.141,149.574
C04442=1131.686,185.145,-62.721,-179.233,9.143,149.574
C04443=1131.682,185.358,-62.742,-179.231,9.146,149.574
C04444=1131.678,185.573,-62.762,-179.229,9.148,149.574
C04445=1131.674,185.788,-62.783,-179.226,9.150,149.574
C04446=1131.670,186.002,-62.804,-179.224,9.153,149.574
C04447=1131.665,186.251,-62.827,-179.221,9.157,149.574
C04448=1131.661,186.500,-62.851,-179.219,9.159,149.574
C04449=1131.656,186.749,-62.875,-179.217,9.162,149.574
C04450=1131.652,186.997,-62.899,-179.214,9.165,149.574
C04451=1131.648,187.246,-62.923,-179.212,9.168,149.574
C04452=1131.643,187.496,-62.947,-179.210,9.170,149.574
C04453=1131.638,187.744,-62.971,-179.207,9.173,149.574
C04454=1131.634,187.993,-62.995,-179.204,9.176,149.574
C04455=1131.629,188.241,-63.019,-179.203,9.179,149.574
C04456=1131.625,188.490,-63.043,-179.200,9.182,149.574
C04457=1131.619,188.739,-63.067,-179.197,9.185,149.574
C04458=1131.616,188.988,-63.091,-179.196,9.187,149.574
C04459=1131.611,189.237,-63.115,-179.193,9.190,149.574
C04460=1131.606,189.486,-63.139,-179.192,9.193,149.575
C04461=1131.602,189.734,-63.163,-179.189,9.196,149.575
C04462=1131.597,189.983,-63.187,-179.187,9.198,149.575
C04463=1131.593,190.231,-63.212,-179.185,9.201,149.575
C04464=1131.588,190.481,-63.235,-179.183,9.204,149.575
C04465=1131.583,190.730,-63.260,-179.181,9.206,149.575
C04466=1131.579,190.978,-63.284,-179.179,9.209,149.575
C04467=1131.575,191.227,-63.308,-179.177,9.212,149.575
C04468=1131.570,191.476,-63.331,-179.175,9.214,149.575
C04469=1131.565,191.725,-63.356,-179.173,9.217,149.575
C04470=1131.561,191.973,-63.381,-179.172,9.219,149.575
C04471=1131.556,192.222,-63.405,-179.169,9.222,149.575
C04472=1131.551,192.471,-63.429,-179.167,9.225,149.575
C04473=1131.547,192.720,-63.453,-179.166,9.228,149.576
C04474=1131.543,192.969,-63.477,-179.164,9.230,149.576
C04475=1131.538,193.217,-63.502,-179.162,9.233,149.576
C04476=1131.533,193.466,-63.526,-179.160,9.235,149.576
C04477=1131.530,193.715,-63.550,-179.159,9.238,149.576
C04478=1131.524,193.964,-63.575,-179.157,9.240,149.576
C04479=1131.520,194.212,-63.599,-179.156,9.243,149.577
C04480=1131.515,194.461,-63.622,-179.154,9.245,149.577
C04481=1131.511,194.711,-63.647,-179.152,9.248,149.577
C04482=1131.506,194.959,-63.671,-179.151,9.250,149.577
C04483=1131.502,195.207,-63.696,-179.150,9.252,149.577
C04484=1131.497,195.456,-63.720,-179.148,9.255,149.577
C04485=1131.493,195.705,-63.745,-179.147,9.257,149.578
C04486=1131.488,195.954,-63.769,-179.145,9.260,149.578
C04487=1131.484,196.202,-63.793,-179.144,9.263,149.578
C04488=1131.480,196.452,-63.818,-179.140,9.266,149.578
C04489=1131.475,196.700,-63.842,-179.136,9.270,149.578
C04490=1131.470,196.949,-63.867,-179.132,9.274,149.577
C04491=1131.466,197.198,-63.892,-179.128,9.278,149.577
C04492=1131.461,197.446,-63.916,-179.124,9.281,149.577
C04493=1131.456,197.695,-63.940,-179.120,9.286,149.577
C04494=1131.452,197.944,-63.965,-179.116,9.289,149.577
C04495=1131.449,198.158,-63.986,-179.113,9.293,149.577
C04496=1131.445,198.373,-64.007,-179.109,9.296,149.577
C04497=1131.440,198.588,-64.028,-179.106,9.299,149.576
C04498=1131.437,198.802,-64.050,-179.103,9.303,149.576
C04499=1131.433,199.016,-64.071,-179.100,9.305,149.576
C04500=1131.429,199.230,-64.092,-179.096,9.309,149.576
C04501=1131.425,199.445,-64.113,-179.093,9.312,149.576
C04502=1131.421,199.659,-64.135,-179.089,9.315,149.576
C04503=1131.416,199.908,-64.159,-179.086,9.319,149.576
C04504=1131.412,200.157,-64.184,-179.082,9.322,149.575
C04505=1131.408,200.405,-64.209,-179.078,9.325,149.575
C04506=1131.403,200.653,-64.234,-179.075,9.329,149.575
C04507=1131.398,200.903,-64.259,-179.072,9.331,149.575
C04508=1131.394,201.151,-64.283,-179.068,9.335,149.575
C04509=1131.390,201.400,-64.308,-179.065,9.338,149.575
C04510=1131.385,201.649,-64.332,-179.061,9.342,149.574
C04511=1131.381,201.897,-64.358,-179.058,9.345,149.574
C04512=1131.376,202.146,-64.383,-179.054,9.348,149.574
C04513=1131.372,202.395,-64.407,-179.051,9.351,149.574
C04514=1131.367,202.643,-64.433,-179.048,9.355,149.574
C04515=1131.363,202.893,-64.458,-179.045,9.357,149.574
C04516=1131.359,203.140,-64.483,-179.041,9.361,149.574
C04517=1131.354,203.390,-64.508,-179.038,9.364,149.573
C04518=1131.349,203.638,-64.533,-179.035,9.367,149.573
C04519=1131.345,203.887,-64.558,-179.032,9.370,149.573
C04520=1131.341,204.135,-64.583,-179.029,9.373,149.573
C04521=1131.336,204.385,-64.608,-179.026,9.376,149.573
C04522=1131.331,204.633,-64.633,-179.023,9.378,149.573
C04523=1131.327,204.882,-64.658,-179.020,9.382,149.573
C04524=1131.322,205.130,-64.684,-179.017,9.385,149.573
C04525=1131.318,205.379,-64.708,-179.014,9.388,149.573
C04526=1131.313,205.628,-64.733,-179.011,9.390,149.572
C04527=1131.309,205.877,-64.758,-179.009,9.392,149.572
C04528=1131.304,206.125,-64.784,-179.007,9.396,149.572
C04529=1131.300,206.374,-64.810,-179.004,9.398,149.572
C04530=1131.294,206.623,-64.834,-179.001,9.401,149.572
C04531=1131.291,206.871,-64.859,-178.998,9.404,149.572
C04532=1131.287,207.120,-64.885,-178.996,9.406,149.572
C04533=1131.282,207.369,-64.910,-178.993,9.409,149.572
C04534=1131.277,207.617,-64.936,-178.991,9.412,149.572
C04535=1131.273,207.866,-64.961,-178.989,9.415,149.572
C04536=1131.268,208.115,-64.986,-178.986,9.417,149.572
C04537=1131.264,208.364,-65.012,-178.984,9.420,149.572
C04538=1131.259,208.612,-65.037,-178.981,9.423,149.572
C04539=1131.254,208.861,-65.062,-178.979,9.425,149.572
C04540=1131.250,209.109,-65.087,-178.977,9.428,149.572
C04541=1131.246,209.358,-65.113,-178.975,9.430,149.572
C04542=1131.242,209.607,-65.138,-178.973,9.433,149.572
C04543=1131.237,209.855,-65.164,-178.970,9.436,149.572
C04544=1131.233,210.104,-65.189,-178.968,9.438,149.572
C04545=1131.228,210.353,-65.215,-178.967,9.440,149.572
C04546=1131.224,210.601,-65.240,-178.965,9.443,149.572
C04547=1131.219,210.850,-65.266,-178.963,9.445,149.572
C04548=1131.215,211.099,-65.292,-178.961,9.448,149.573
C04549=1131.210,211.347,-65.316,-178.959,9.450,149.573
C04550=1131.206,211.596,-65.342,-178.958,9.453,149.573
C04551=1131.201,211.811,-65.364,-178.956,9.455,149.573
C04552=1131.198,212.024,-65.386,-178.954,9.457,149.573
C04553=1131.194,212.239,-65.409,-178.953,9.459,149.573
C04554=1131.191,212.453,-65.430,-178.951,9.462,149.573
C04555=1131.186,212.667,-65.452,-178.951,9.464,149.573
C04556=1131.182,212.881,-65.474,-178.949,9.465,149.573
C04557=1131.179,213.096,-65.496,-178.948,9.468,149.574
C04558=1131.175,213.310,-65.518,-178.947,9.469,149.574
C04559=1131.170,213.559,-65.544,-178.945,9.472,149.574
C04560=1131.166,213.807,-65.569,-178.944,9.475,149.574
C04561=1131.161,214.056,-65.595,-178.941,9.478,149.574
C04562=1131.157,214.305,-65.621,-178.940,9.481,149.574
C04563=1131.152,214.553,-65.646,-178.938,9.483,149.575
C04564=1131.148,214.802,-65.672,-178.936,9.486,149.575
C04565=1131.144,215.051,-65.698,-178.934,9.489,149.575
C04566=1131.140,215.299,-65.723,-178.932,9.491,149.575
C04567=1131.135,215.547,-65.749,-178.930,9.494,149.575
C04568=1131.131,215.796,-65.775,-178.928,9.497,149.575
C04569=1131.126,216.045,-65.800,-178.926,9.500,149.575
C04570=1131.121,216.293,-65.826,-178.924,9.503,149.575
C04571=1131.117,216.542,-65.852,-178.922,9.505,149.576
C04572=1131.112,216.791,-65.878,-178.920,9.508,149.576
C04573=1131.108,217.040,-65.904,-178.918,9.511,149.576
C04574=1131.104,217.288,-65.930,-178.916,9.514,149.576
C04575=1131.099,217.536,-65.955,-178.913,9.517,149.576
C04576=1131.095,217.785,-65.981,-178.911,9.520,149.576
C04577=1131.090,218.034,-66.008,-178.909,9.523,149.576
C04578=1131.086,218.283,-66.033,-178.907,9.526,149.577
C04579=1131.081,218.531,-66.059,-178.904,9.529,149.577
C04580=1131.077,218.780,-66.084,-178.902,9.532,149.577
C04581=1131.073,219.029,-66.110,-178.900,9.535,149.577
C04582=1131.069,219.277,-66.137,-178.898,9.538,149.577
C04583=1131.064,219.526,-66.163,-178.895,9.541,149.577
C04584=1131.059,219.774,-66.188,-178.893,9.544,149.577
C04585=1131.055,220.023,-66.214,-178.890,9.548,149.577
C04586=1131.051,220.271,-66.241,-178.888,9.551,149.577
C04587=1131.046,220.520,-66.267,-178.885,9.554,149.577
C04588=1131.042,220.769,-66.293,-178.883,9.557,149.577
C04589=1131.037,221.018,-66.318,-178.880,9.560,149.577
C04590=1131.033,221.265,-66.345,-178.877,9.563,149.577
C04591=1131.028,221.514,-66.371,-178.874,9.567,149.578
C04592=1131.024,221.763,-66.397,-178.872,9.570,149.578
C04593=1131.020,222.011,-66.423,-178.869,9.573,149.578
C04594=1131.015,222.260,-66.449,-178.867,9.576,149.578
C04595=1131.011,222.509,-66.475,-178.864,9.580,149.578
C04596=1131.006,222.757,-66.501,-178.861,9.583,149.578
C04597=1131.001,223.006,-66.528,-178.858,9.586,149.578
C04598=1130.997,223.255,-66.553,-178.855,9.590,149.578
C04599=1130.993,223.503,-66.580,-178.852,9.593,149.578
C04600=1130.988,223.752,-66.606,-178.849,9.597,149.578
C04601=1130.984,224.000,-66.633,-178.846,9.600,149.578
C04602=1130.980,224.249,-66.658,-178.843,9.603,149.578
C04603=1130.975,224.497,-66.686,-178.840,9.606,149.578
C04604=1130.971,224.746,-66.711,-178.837,9.610,149.578
C04605=1130.966,224.995,-66.738,-178.833,9.614,149.578
C04606=1130.962,225.244,-66.764,-178.830,9.616,149.578
C04607=1130.958,225.457,-66.787,-178.828,9.620,149.578
C04608=1130.954,225.671,-66.810,-178.825,9.622,149.577
C04609=1130.950,225.886,-66.832,-178.822,9.625,149.578
C04610=1130.946,226.099,-66.855,-178.819,9.629,149.577
C04611=1130.943,226.314,-66.878,-178.816,9.632,149.577
C04612=1130.939,226.527,-66.901,-178.813,9.635,149.577
C04613=1130.935,226.742,-66.923,-178.810,9.638,149.577
C04614=1130.931,226.956,-66.946,-178.808,9.640,149.577
C04615=1130.927,227.204,-66.973,-178.804,9.644,149.577
C04616=1130.922,227.453,-67.000,-178.801,9.648,149.577
C04617=1130.918,227.702,-67.025,-178.797,9.651,149.577
C04618=1130.914,227.950,-67.052,-178.794,9.655,149.577
C04619=1130.910,228.198,-67.079,-178.790,9.658,149.577
C04620=1130.905,228.447,-67.105,-178.786,9.662,149.577
C04621=1130.901,228.696,-67.132,-178.783,9.665,149.576
C04622=1130.896,228.944,-67.159,-178.779,9.668,149.576
C04623=1130.891,229.193,-67.186,-178.775,9.672,149.576
C04624=1130.888,229.441,-67.212,-178.772,9.675,149.576
C04625=1130.883,229.691,-67.239,-178.768,9.679,149.576
C04626=1130.879,229.939,-67.266,-178.764,9.682,149.576
C04627=1130.875,230.187,-67.293,-178.760,9.686,149.575
C04628=1130.870,230.436,-67.320,-178.756,9.690,149.575
C04629=1130.865,230.684,-67.347,-178.752,9.693,149.575
C04630=1130.861,230.932,-67.373,-178.749,9.697,149.575
C04631=1130.857,231.181,-67.400,-178.745,9.700,149.575
C04632=1130.852,231.429,-67.427,-178.742,9.703,149.574
C04633=1130.848,231.678,-67.454,-178.738,9.706,149.574
C04634=1130.843,231.926,-67.481,-178.735,9.710,149.574
C04635=1130.839,232.175,-67.508,-178.731,9.713,149.574
C04636=1130.836,232.423,-67.535,-178.728,9.716,149.574
C04637=1130.831,232.672,-67.562,-178.724,9.719,149.574
C04638=1130.826,232.920,-67.589,-178.721,9.722,149.574
C04639=1130.822,233.169,-67.616,-178.718,9.725,149.573
C04640=1130.817,233.417,-67.643,-178.715,9.728,149.573
C04641=1130.813,233.666,-67.669,-178.711,9.732,149.573
C04642=1130.809,233.915,-67.697,-178.708,9.734,149.573
C04643=1130.804,234.163,-67.724,-178.705,9.737,149.573
C04644=1130.800,234.412,-67.751,-178.702,9.739,149.573
C04645=1130.795,234.660,-67.778,-178.698,9.743,149.572
C04646=1130.791,234.908,-67.804,-178.695,9.746,149.572
C04647=1130.787,235.157,-67.833,-178.692,9.748,149.572
C04648=1130.783,235.406,-67.860,-178.689,9.751,149.572
C04649=1130.778,235.654,-67.887,-178.686,9.754,149.572
C04650=1130.773,235.903,-67.914,-178.683,9.757,149.572
C04651=1130.769,236.151,-67.941,-178.681,9.759,149.572
C04652=1130.765,236.400,-67.969,-178.678,9.763,149.572
C04653=1130.760,236.648,-67.996,-178.675,9.765,149.572
C04654=1130.756,236.896,-68.022,-178.672,9.768,149.572
C04655=1130.752,237.144,-68.050,-178.670,9.770,149.571
C04656=1130.748,237.393,-68.078,-178.667,9.773,149.571
C04657=1130.743,237.642,-68.105,-178.664,9.776,149.571
C04658=1130.739,237.890,-68.132,-178.661,9.779,149.571
C04659=1130.734,238.138,-68.160,-178.659,9.781,149.571
C04660=1130.730,238.387,-68.187,-178.656,9.783,149.571
C04661=1130.726,238.635,-68.215,-178.654,9.785,149.571
C04662=1130.721,238.884,-68.242,-178.651,9.788,149.571
C04663=1130.718,239.098,-68.265,-178.649,9.790,149.571
C04664=1130.714,239.312,-68.289,-178.647,9.793,149.571
C04665=1130.710,239.526,-68.312,-178.645,9.795,149.571
C04666=1130.706,239.740,-68.337,-178.643,9.797,149.571
C04667=1130.703,239.954,-68.360,-178.641,9.798,149.571
C04668=1130.699,240.168,-68.384,-178.639,9.801,149.571
C04669=1130.695,240.382,-68.407,-178.637,9.803,149.571
C04670=1130.691,240.596,-68.431,-178.635,9.805,149.571
C04671=1130.687,240.844,-68.458,-178.633,9.807,149.571
C04672=1130.683,241.093,-68.486,-178.631,9.810,149.571
C04673=1130.678,241.341,-68.513,-178.629,9.811,149.570
C04674=1130.673,241.589,-68.542,-178.627,9.814,149.571
C04675=1130.669,241.839,-68.569,-178.625,9.816,149.571
C04676=1130.665,242.087,-68.597,-178.623,9.818,149.571
C04677=1130.660,242.335,-68.624,-178.621,9.820,149.571
C04678=1130.656,242.584,-68.652,-178.619,9.823,149.571
C04679=1130.652,242.832,-68.679,-178.617,9.825,149.571
C04680=1130.647,243.080,-68.707,-178.615,9.827,149.571
C04681=1130.643,243.329,-68.734,-178.613,9.830,149.571
C04682=1130.639,243.577,-68.762,-178.612,9.831,149.571
C04683=1130.635,243.825,-68.790,-178.610,9.834,149.571
C04684=1130.631,244.074,-68.817,-178.609,9.836,149.571
C04685=1130.626,244.322,-68.846,-178.607,9.839,149.571
C04686=1130.622,244.572,-68.873,-178.606,9.840,149.571
C04687=1130.617,244.819,-68.901,-178.604,9.843,149.571
C04688=1130.613,245.067,-68.929,-178.603,9.845,149.571
C04689=1130.609,245.316,-68.956,-178.601,9.847,149.572
C04690=1130.604,245.564,-68.984,-178.600,9.849,149.572
C04691=1130.601,245.813,-69.012,-178.598,9.851,149.572
C04692=1130.595,246.062,-69.040,-178.597,9.853,149.572
C04693=1130.591,246.310,-69.067,-178.595,9.855,149.572
C04694=1130.587,246.558,-69.096,-178.595,9.857,149.572
C04695=1130.583,246.807,-69.123,-178.594,9.859,149.573
C04696=1130.578,247.055,-69.150,-178.592,9.862,149.573
C04697=1130.574,247.303,-69.179,-178.591,9.863,149.573
C04698=1130.569,247.552,-69.206,-178.586,9.867,149.573
C04699=1130.565,247.800,-69.234,-178.579,9.873,149.572
C04700=1130.561,248.048,-69.262,-178.572,9.879,149.572
C04701=1130.557,248.297,-69.290,-178.565,9.884,149.571
C04702=1130.552,248.546,-69.318,-178.558,9.889,149.570
C04703=1130.548,248.794,-69.346,-178.552,9.894,149.570
C04704=1130.544,249.042,-69.374,-178.546,9.898,149.569
C04705=1130.539,249.290,-69.402,-178.539,9.903,149.569
C04706=1130.535,249.539,-69.430,-178.534,9.908,149.568
C04707=1130.531,249.788,-69.459,-178.529,9.911,149.568
C04708=1130.526,250.036,-69.487,-178.523,9.916,149.567
C04709=1130.522,250.284,-69.515,-178.518,9.920,149.567
C04710=1130.518,250.532,-69.543,-178.513,9.923,149.567
C04711=1130.513,250.781,-69.572,-178.509,9.926,149.566
C04712=1130.509,251.029,-69.599,-178.505,9.930,149.566
C04713=1130.505,251.278,-69.628,-178.501,9.933,149.566
C04714=1130.500,251.526,-69.656,-178.497,9.936,149.566
C04715=1130.496,251.775,-69.685,-178.494,9.938,149.565
C04716=1130.492,252.023,-69.713,-178.491,9.941,149.565
C04717=1130.488,252.270,-69.741,-178.488,9.944,149.565
C04718=1130.483,252.519,-69.770,-178.485,9.946,149.565
C04719=1130.480,252.733,-69.794,-178.483,9.947,149.565
C04720=1130.476,252.947,-69.819,-178.481,9.950,149.565
C04721=1130.473,253.161,-69.843,-178.479,9.951,149.564
C04722=1130.469,253.375,-69.867,-178.478,9.953,149.564
C04723=1130.465,253.589,-69.892,-178.477,9.954,149.565
C04724=1130.461,253.803,-69.917,-178.476,9.956,149.565
C04725=1130.457,254.017,-69.941,-178.474,9.957,149.565
C04726=1130.454,254.231,-69.966,-178.474,9.958,149.565
C04727=1130.449,254.478,-69.994,-178.474,9.959,149.565
C04728=1130.445,254.727,-70.023,-178.473,9.960,149.565
C04729=1130.441,254.975,-70.051,-178.473,9.961,149.565
C04730=1130.436,255.224,-70.080,-178.473,9.962,149.565
C04731=1130.432,255.472,-70.108,-178.474,9.963,149.566
C04732=1130.428,255.720,-70.137,-178.475,9.963,149.566
C04733=1130.424,255.968,-70.165,-178.475,9.964,149.566
C04734=1130.419,256.217,-70.194,-178.472,9.967,149.567
C04735=1130.415,256.465,-70.221,-178.469,9.970,149.566
C04736=1130.411,256.713,-70.251,-178.467,9.973,149.566
C04737=1130.407,256.961,-70.279,-178.464,9.976,149.566
C04738=1130.402,257.210,-70.307,-178.461,9.978,149.566
C04739=1130.398,257.459,-70.336,-178.458,9.981,149.566
C04740=1130.393,257.706,-70.365,-178.455,9.984,149.566
C04741=1130.389,257.955,-70.393,-178.451,9.988,149.566
C04742=1130.385,258.204,-70.422,-178.448,9.990,149.566
C04743=1130.380,258.451,-70.451,-178.445,9.993,149.566
C04744=1130.376,258.700,-70.479,-178.442,9.996,149.565
C04745=1130.373,258.948,-70.508,-178.439,9.999,149.565
C04746=1130.367,259.196,-70.537,-178.436,10.002,149.565
C04747=1130.363,259.445,-70.565,-178.432,10.006,149.565
C04748=1130.360,259.693,-70.594,-178.429,10.008,149.565
C04749=1130.355,259.942,-70.623,-178.425,10.012,149.565
C04750=1130.350,260.190,-70.652,-178.422,10.014,149.565
C04751=1130.346,260.438,-70.680,-178.419,10.018,149.565
C04752=1130.342,260.687,-70.710,-178.415,10.020,149.564
C04753=1130.337,260.935,-70.738,-178.412,10.024,149.564
C04754=1130.334,261.183,-70.767,-178.409,10.027,149.564
C04755=1130.329,261.432,-70.796,-178.405,10.030,149.564
C04756=1130.325,261.680,-70.825,-178.401,10.033,149.564
C04757=1130.320,261.928,-70.853,-178.398,10.036,149.563
C04758=1130.317,262.176,-70.882,-178.394,10.039,149.563
C04759=1130.312,262.424,-70.912,-178.390,10.042,149.563
C04760=1130.308,262.673,-70.940,-178.386,10.045,149.563
C04761=1130.304,262.921,-70.970,-178.384,10.048,149.563
C04762=1130.299,263.169,-70.999,-178.380,10.051,149.562
C04763=1130.295,263.418,-71.027,-178.376,10.055,149.562
C04764=1130.291,263.666,-71.057,-178.372,10.058,149.562
C04765=1130.287,263.914,-71.086,-178.368,10.061,149.562
C04766=1130.282,264.163,-71.115,-178.364,10.064,149.561
C04767=1130.278,264.411,-71.144,-178.360,10.068,149.561
C04768=1130.273,264.659,-71.173,-178.357,10.070,149.561
C04769=1130.269,264.907,-71.203,-178.355,10.072,149.561
C04770=1130.265,265.156,-71.231,-178.352,10.074,149.561
C04771=1130.261,265.404,-71.260,-178.350,10.076,149.561
C04772=1130.257,265.652,-71.290,-178.347,10.079,149.561
C04773=1130.252,265.900,-71.319,-178.345,10.081,149.560
C04774=1130.248,266.148,-71.348,-178.342,10.084,149.561
C04775=1130.245,266.361,-71.374,-178.340,10.086,149.560
C04776=1130.241,266.576,-71.399,-178.338,10.088,149.560
C04777=1130.237,266.790,-71.424,-178.335,10.090,149.560
C04778=1130.233,267.003,-71.449,-178.334,10.092,149.560
C04779=1130.230,267.217,-71.474,-178.331,10.094,149.560
C04780=1130.226,267.431,-71.499,-178.329,10.096,149.560
C04781=1130.222,267.645,-71.525,-178.327,10.098,149.560
C04782=1130.219,267.859,-71.550,-178.325,10.101,149.560
C04783=1130.215,268.107,-71.580,-178.322,10.103,149.560
C04784=1130.210,268.355,-71.609,-178.320,10.106,149.560
C04785=1130.206,268.603,-71.639,-178.317,10.107,149.560
C04786=1130.201,268.851,-71.668,-178.314,10.110,149.559
C04787=1130.197,269.099,-71.697,-178.311,10.113,149.559
C04788=1130.193,269.348,-71.727,-178.309,10.115,149.559
C04789=1130.189,269.596,-71.756,-178.306,10.118,149.559
C04790=1130.185,269.844,-71.786,-178.303,10.120,149.559
C04791=1130.180,270.092,-71.815,-178.301,10.122,149.559
C04792=1130.176,270.341,-71.844,-178.298,10.125,149.559
C04793=1130.172,270.589,-71.874,-178.295,10.128,149.559
C04794=1130.168,270.837,-71.903,-178.292,10.131,149.559
C04795=1130.164,271.085,-71.933,-178.289,10.134,149.558
C04796=1130.160,271.334,-71.962,-178.287,10.135,149.558
C04797=1130.155,271.582,-71.992,-178.284,10.138,149.558
C04798=1130.151,271.830,-72.022,-178.281,10.141,149.558
C04799=1130.147,272.078,-72.052,-178.278,10.144,149.558
C04800=1130.142,272.326,-72.081,-178.275,10.147,149.558
C04801=1130.138,272.575,-72.111,-178.272,10.149,149.558
C04802=1130.134,272.823,-72.140,-178.269,10.152,149.558
C04803=1130.130,273.071,-72.170,-178.266,10.154,149.557
C04804=1130.126,273.319,-72.200,-178.263,10.157,149.557
C04805=1130.121,273.567,-72.230,-178.260,10.160,149.557
C04806=1130.117,273.816,-72.259,-178.257,10.163,149.557
C04807=1130.113,274.064,-72.289,-178.254,10.165,149.557
C04808=1130.109,274.312,-72.319,-178.251,10.168,149.557
C04809=1130.105,274.560,-72.348,-178.248,10.171,149.557
C04810=1130.100,274.808,-72.378,-178.245,10.173,149.557
C04811=1130.096,275.057,-72.408,-178.242,10.176,149.556
C04812=1130.092,275.304,-72.438,-178.239,10.179,149.556
C04813=1130.087,275.553,-72.468,-178.236,10.181,149.556
C04814=1130.083,275.801,-72.497,-178.233,10.184,149.556
C04815=1130.079,276.049,-72.528,-178.230,10.187,149.556
C04816=1130.075,276.297,-72.557,-178.226,10.190,149.556
C04817=1130.071,276.545,-72.587,-178.223,10.193,149.556
C04818=1130.067,276.794,-72.617,-178.219,10.195,149.555
C04819=1130.062,277.042,-72.647,-178.216,10.198,149.555
C04820=1130.058,277.290,-72.678,-178.213,10.202,149.555
C04821=1130.054,277.538,-72.707,-178.210,10.204,149.555
C04822=1130.049,277.786,-72.738,-178.207,10.207,149.555
C04823=1130.045,278.035,-72.767,-178.203,10.209,149.554
C04824=1130.041,278.282,-72.797,-178.200,10.213,149.554
C04825=1130.036,278.531,-72.827,-178.196,10.215,149.554
C04826=1130.033,278.779,-72.858,-178.193,10.217,149.554
C04827=1130.029,279.027,-72.887,-178.189,10.221,149.554
C04828=1130.024,279.275,-72.918,-178.186,10.223,149.553
C04829=1130.021,279.523,-72.948,-178.183,10.226,149.553
C04830=1130.016,279.772,-72.978,-178.179,10.229,149.553
C04831=1130.013,279.985,-73.005,-178.176,10.232,149.553
C04832=1130.009,280.199,-73.030,-178.174,10.234,149.553
C04833=1130.005,280.412,-73.056,-178.171,10.237,149.553
C04834=1130.002,280.626,-73.082,-178.167,10.239,149.552
C04835=1129.997,280.840,-73.108,-178.164,10.242,149.552
C04836=1129.995,281.053,-73.134,-178.161,10.244,149.552
C04837=1129.991,281.266,-73.161,-178.158,10.247,149.552
C04838=1129.987,281.480,-73.186,-178.155,10.249,149.551
C04839=1129.983,281.728,-73.217,-178.152,10.251,149.551
C04840=1129.979,281.977,-73.247,-178.149,10.254,149.551
C04841=1129.974,282.225,-73.277,-178.146,10.256,149.551
C04842=1129.971,282.472,-73.308,-178.143,10.259,149.551
C04843=1129.966,282.721,-73.339,-178.140,10.262,149.551
C04844=1129.962,282.969,-73.370,-178.136,10.264,149.550
C04845=1129.958,283.217,-73.399,-178.134,10.267,149.550
C04846=1129.953,283.465,-73.430,-178.131,10.270,149.550
C04847=1129.949,283.713,-73.460,-178.127,10.272,149.550
C04848=1129.945,283.961,-73.491,-178.124,10.275,149.550
C04849=1129.941,284.209,-73.521,-178.121,10.277,149.549
C04850=1129.937,284.457,-73.552,-178.119,10.279,149.549
C04851=1129.933,284.706,-73.582,-178.115,10.282,149.549
C04852=1129.929,284.954,-73.613,-178.112,10.284,149.549
C04853=1129.924,285.202,-73.643,-178.109,10.287,149.549
C04854=1129.920,285.450,-73.674,-178.106,10.289,149.549
C04855=1129.916,285.698,-73.705,-178.103,10.292,149.548
C04856=1129.911,285.946,-73.735,-178.100,10.295,149.548
C04857=1129.908,286.194,-73.766,-178.097,10.297,149.548
C04858=1129.904,286.443,-73.797,-178.094,10.300,149.548
C04859=1129.899,286.690,-73.827,-178.091,10.303,149.548
C04860=1129.895,286.938,-73.858,-178.088,10.304,149.547
C04861=1129.891,287.187,-73.889,-178.085,10.307,149.547
C04862=1129.886,287.435,-73.920,-178.082,10.310,149.547
C04863=1129.883,287.682,-73.950,-178.079,10.312,149.547
C04864=1129.879,287.931,-73.981,-178.076,10.315,149.547
C04865=1129.874,288.179,-74.012,-178.072,10.317,149.547
C04866=1129.870,288.427,-74.042,-178.069,10.320,149.547
C04867=1129.866,288.675,-74.073,-178.066,10.323,149.546
C04868=1129.862,288.923,-74.104,-178.063,10.325,149.546
C04869=1129.857,289.171,-74.135,-178.060,10.328,149.546
C04870=1129.854,289.419,-74.166,-178.057,10.331,149.546
C04871=1129.849,289.667,-74.196,-178.054,10.332,149.545
C04872=1129.845,289.915,-74.227,-178.051,10.335,149.545
C04873=1129.841,290.164,-74.258,-178.048,10.338,149.545
C04874=1129.837,290.411,-74.289,-178.045,10.340,149.545
C04875=1129.833,290.659,-74.320,-178.042,10.343,149.545
C04876=1129.828,290.907,-74.351,-178.039,10.345,149.545
C04877=1129.824,291.156,-74.382,-178.036,10.348,149.545
C04878=1129.820,291.403,-74.414,-178.032,10.350,149.544
C04879=1129.816,291.651,-74.444,-178.030,10.353,149.544
C04880=1129.812,291.899,-74.475,-178.026,10.356,149.544
C04881=1129.808,292.147,-74.506,-178.023,10.358,149.544
C04882=1129.804,292.395,-74.538,-178.020,10.361,149.544
C04883=1129.799,292.643,-74.568,-178.018,10.363,149.543
C04884=1129.795,292.892,-74.600,-178.014,10.365,149.543
C04885=1129.791,293.139,-74.631,-178.011,10.368,149.543
C04886=1129.788,293.388,-74.662,-178.008,10.370,149.543
C04887=1129.784,293.601,-74.688,-178.005,10.373,149.543
C04888=1129.780,293.815,-74.715,-178.003,10.375,149.543
C04889=1129.777,294.027,-74.742,-178.000,10.377,149.542
C04890=1129.773,294.241,-74.769,-177.997,10.380,149.542
C04891=1129.770,294.455,-74.796,-177.995,10.382,149.542
C04892=1129.766,294.668,-74.822,-177.993,10.384,149.542
C04893=1129.762,294.882,-74.849,-177.990,10.386,149.542
C04894=1129.759,295.095,-74.877,-177.987,10.388,149.542
C04895=1129.755,295.343,-74.908,-177.984,10.391,149.542
C04896=1129.751,295.591,-74.939,-177.981,10.393,149.541
C04897=1129.746,295.839,-74.970,-177.978,10.396,149.541
C04898=1129.743,296.087,-75.002,-177.974,10.398,149.541
C04899=1129.738,296.335,-75.033,-177.971,10.401,149.541
C04900=1129.734,296.583,-75.065,-177.968,10.404,149.541
C04901=1129.730,296.831,-75.095,-177.965,10.406,149.540
C04902=1129.726,297.079,-75.127,-177.962,10.409,149.540
C04903=1129.721,297.327,-75.158,-177.959,10.411,149.540
C04904=1129.718,297.575,-75.190,-177.956,10.413,149.540
C04905=1129.713,297.823,-75.222,-177.953,10.416,149.540
C04906=1129.709,298.071,-75.253,-177.950,10.418,149.539
C04907=1129.705,298.319,-75.285,-177.947,10.421,149.539
C04908=1129.701,298.567,-75.316,-177.944,10.424,149.539
C04909=1129.697,298.815,-75.347,-177.941,10.426,149.539
C04910=1129.692,299.063,-75.379,-177.937,10.429,149.539
C04911=1129.689,299.311,-75.411,-177.934,10.432,149.539
C04912=1129.685,299.559,-75.442,-177.931,10.434,149.538
C04913=1129.680,299.807,-75.473,-177.928,10.437,149.538
C04914=1129.677,300.055,-75.505,-177.925,10.439,149.538
C04915=1129.672,300.302,-75.537,-177.922,10.442,149.538
C04916=1129.668,300.551,-75.568,-177.919,10.444,149.538
C04917=1129.664,300.799,-75.600,-177.916,10.446,149.538
C04918=1129.659,301.046,-75.632,-177.913,10.449,149.537
C04919=1129.656,301.294,-75.664,-177.910,10.452,149.537
C04920=1129.652,301.542,-75.695,-177.907,10.454,149.537
C04921=1129.647,301.790,-75.728,-177.904,10.457,149.537
C04922=1129.643,302.039,-75.759,-177.900,10.459,149.537
C04923=1129.639,302.286,-75.790,-177.897,10.462,149.537
C04924=1129.635,302.534,-75.822,-177.894,10.464,149.536
C04925=1129.631,302.783,-75.854,-177.891,10.467,149.536
C04926=1129.626,303.030,-75.886,-177.888,10.470,149.536
C04927=1129.623,303.278,-75.918,-177.885,10.472,149.536
C04928=1129.619,303.526,-75.950,-177.882,10.475,149.536
C04929=1129.614,303.774,-75.982,-177.878,10.477,149.535
C04930=1129.610,304.022,-76.014,-177.876,10.479,149.535
C04931=1129.606,304.270,-76.045,-177.873,10.482,149.535
C04932=1129.602,304.518,-76.078,-177.870,10.484,149.535
C04933=1129.598,304.765,-76.109,-177.866,10.487,149.535
C04934=1129.594,305.013,-76.141,-177.863,10.490,149.535
C04935=1129.589,305.262,-76.174,-177.860,10.492,149.534
C04936=1129.585,305.509,-76.205,-177.857,10.495,149.534
C04937=1129.581,305.757,-76.237,-177.854,10.497,149.534
C04938=1129.577,306.005,-76.269,-177.850,10.500,149.534
C04939=1129.573,306.253,-76.301,-177.848,10.502,149.534
C04940=1129.569,306.501,-76.333,-177.844,10.505,149.533
C04941=1129.565,306.749,-76.365,-177.841,10.508,149.533
C04942=1129.561,306.997,-76.398,-177.838,10.510,149.533
C04943=1129.557,307.211,-76.425,-177.836,10.512,149.533
C04944=1129.553,307.423,-76.452,-177.833,10.514,149.533
C04945=1129.550,307.636,-76.480,-177.830,10.516,149.532
C04946=1129.546,307.850,-76.508,-177.828,10.518,149.532
C04947=1129.543,308.063,-76.536,-177.824,10.521,149.532
C04948=1129.540,308.277,-76.564,-177.822,10.523,149.532
C04949=1129.536,308.490,-76.591,-177.820,10.525,149.532
C04950=1129.533,308.704,-76.618,-177.816,10.527,149.532
C04951=1129.528,308.951,-76.651,-177.814,10.530,149.532
C04952=1129.525,309.199,-76.683,-177.810,10.533,149.531
C04953=1129.520,309.447,-76.715,-177.807,10.535,149.531
C04954=1129.517,309.694,-76.748,-177.805,10.537,149.531
C04955=1129.512,309.943,-76.780,-177.802,10.540,149.531
C04956=1129.509,310.191,-76.812,-177.798,10.542,149.531
C04957=1129.504,310.438,-76.845,-177.795,10.545,149.530
C04958=1129.500,310.686,-76.877,-177.792,10.547,149.530
C04959=1129.496,310.934,-76.909,-177.789,10.550,149.530
C04960=1129.492,311.182,-76.942,-177.786,10.553,149.530
C04961=1129.488,311.430,-76.974,-177.782,10.555,149.530
C04962=1129.484,311.678,-77.006,-177.780,10.558,149.530
C04963=1129.479,311.925,-77.039,-177.776,10.560,149.529
C04964=1129.475,312.173,-77.071,-177.773,10.563,149.529
C04965=1129.472,312.421,-77.104,-177.770,10.565,149.529
C04966=1129.467,312.669,-77.136,-177.767,10.568,149.529
C04967=1129.464,312.917,-77.169,-177.764,10.571,149.529
C04968=1129.459,313.165,-77.201,-177.760,10.573,149.528
C04969=1129.455,313.413,-77.234,-177.757,10.575,149.528
C04970=1129.451,313.661,-77.266,-177.755,10.577,149.528
C04971=1129.447,313.908,-77.299,-177.751,10.580,149.528
C04972=1129.443,314.156,-77.331,-177.748,10.583,149.528
C04973=1129.439,314.404,-77.364,-177.745,10.585,149.528
C04974=1129.434,314.652,-77.397,-177.742,10.588,149.527
C04975=1129.431,314.899,-77.429,-177.739,10.590,149.527
C04976=1129.427,315.147,-77.462,-177.736,10.593,149.527
C04977=1129.422,315.395,-77.495,-177.733,10.596,149.527
C04978=1129.419,315.643,-77.527,-177.729,10.598,149.527
C04979=1129.415,315.891,-77.560,-177.726,10.600,149.526
C04980=1129.410,316.139,-77.593,-177.723,10.603,149.526
C04981=1129.406,316.387,-77.626,-177.720,10.606,149.526
C04982=1129.403,316.634,-77.659,-177.716,10.608,149.526
C04983=1129.398,316.882,-77.691,-177.713,10.611,149.526
C04984=1129.394,317.130,-77.724,-177.710,10.613,149.525
C04985=1129.391,317.378,-77.757,-177.707,10.616,149.525
C04986=1129.387,317.625,-77.790,-177.704,10.619,149.525
C04987=1129.382,317.874,-77.822,-177.701,10.621,149.525
C04988=1129.378,318.121,-77.855,-177.698,10.623,149.525
C04989=1129.375,318.369,-77.888,-177.695,10.625,149.525
C04990=1129.371,318.616,-77.921,-177.692,10.628,149.524
C04991=1129.367,318.864,-77.954,-177.689,10.631,149.524
C04992=1129.362,319.113,-77.987,-177.685,10.633,149.524
C04993=1129.358,319.360,-78.020,-177.682,10.635,149.524
C04994=1129.354,319.608,-78.053,-177.679,10.638,149.524
C04995=1129.350,319.855,-78.086,-177.676,10.641,149.523
C04996=1129.346,320.103,-78.119,-177.673,10.643,149.523
C04997=1129.342,320.351,-78.152,-177.670,10.646,149.523
C04998=1129.338,320.599,-78.185,-177.666,10.648,149.523
C04999=1129.334,320.812,-78.213,-177.664,10.650,149.523
C05000=1129.332,321.025,-78.242,-177.661,10.653,149.522
C05001=1129.328,321.239,-78.270,-177.658,10.655,149.522
C05002=1129.325,321.452,-78.299,-177.655,10.658,149.522
C05003=1129.321,321.665,-78.328,-177.653,10.659,149.522
C05004=1129.317,321.878,-78.356,-177.650,10.661,149.522
C05005=1129.314,322.091,-78.384,-177.647,10.664,149.522
C05006=1129.311,322.304,-78.413,-177.645,10.666,149.522
C05007=1129.307,322.552,-78.446,-177.641,10.668,149.521
C05008=1129.302,322.800,-78.479,-177.639,10.671,149.521
C05009=1129.298,323.047,-78.512,-177.635,10.673,149.521
C05010=1129.295,323.295,-78.546,-177.632,10.676,149.521
C05011=1129.291,323.543,-78.579,-177.629,10.678,149.520
C05012=1129.287,323.791,-78.613,-177.626,10.681,149.520
C05013=1129.283,324.038,-78.646,-177.622,10.683,149.520
C05014=1129.278,324.286,-78.679,-177.619,10.686,149.520
C05015=1129.274,324.534,-78.712,-177.616,10.689,149.520
C05016=1129.270,324.782,-78.745,-177.613,10.691,149.520
C05017=1129.267,325.029,-78.779,-177.609,10.694,149.519
C05018=1129.263,325.277,-78.813,-177.607,10.696,149.519
C05019=1129.259,325.525,-78.846,-177.604,10.698,149.519
C05020=1129.255,325.773,-78.879,-177.600,10.700,149.519
C05021=1129.250,326.020,-78.912,-177.598,10.703,149.519
C05022=1129.247,326.267,-78.946,-177.594,10.706,149.518
C05023=1129.243,326.516,-78.979,-177.591,10.708,149.518
C05024=1129.239,326.764,-79.013,-177.588,10.711,149.518
C05025=1129.235,327.011,-79.046,-177.585,10.713,149.518
C05026=1129.231,327.258,-79.080,-177.581,10.716,149.518
C05027=1129.226,327.507,-79.113,-177.578,10.718,149.517
C05028=1129.223,327.755,-79.147,-177.575,10.721,149.517
C05029=1129.219,328.002,-79.181,-177.572,10.723,149.517
C05030=1129.215,328.250,-79.214,-177.568,10.726,149.517
C05031=1129.211,328.497,-79.248,-177.566,10.729,149.517
C05032=1129.207,328.745,-79.281,-177.562,10.731,149.517
C05033=1129.203,328.993,-79.314,-177.559,10.734,149.516
C05034=1129.198,329.240,-79.349,-177.556,10.736,149.516
C05035=1129.194,329.488,-79.382,-177.553,10.739,149.516
C05036=1129.190,329.735,-79.416,-177.549,10.741,149.516
C05037=1129.187,329.984,-79.449,-177.546,10.744,149.516
C05038=1129.183,330.231,-79.483,-177.543,10.746,149.515
C05039=1129.178,330.479,-79.517,-177.540,10.749,149.515
C05040=1129.175,330.727,-79.551,-177.537,10.751,149.515
C05041=1129.171,330.974,-79.584,-177.534,10.753,149.515
C05042=1129.167,331.222,-79.618,-177.531,10.756,149.515
C05043=1129.162,331.470,-79.652,-177.527,10.758,149.514
C05044=1129.159,331.717,-79.686,-177.524,10.761,149.514
C05045=1129.155,331.965,-79.719,-177.521,10.763,149.514
C05046=1129.150,332.213,-79.754,-177.518,10.766,149.514
C05047=1129.147,332.460,-79.788,-177.515,10.768,149.514
C05048=1129.143,332.708,-79.821,-177.511,10.771,149.513
C05049=1129.139,332.955,-79.855,-177.508,10.774,149.513
C05050=1129.135,333.204,-79.889,-177.505,10.776,149.513
C05051=1129.131,333.451,-79.923,-177.502,10.779,149.513
C05052=1129.127,333.698,-79.957,-177.498,10.781,149.513
C05053=1129.123,333.946,-79.992,-177.495,10.784,149.513
C05054=1129.119,334.194,-80.025,-177.492,10.786,149.512
C05055=1129.115,334.407,-80.054,-177.489,10.788,149.512
C05056=1129.113,334.620,-80.084,-177.487,10.791,149.512
C05057=1129.109,334.833,-80.113,-177.484,10.792,149.512
C05058=1129.105,335.046,-80.142,-177.482,10.794,149.512
C05059=1129.102,335.260,-80.172,-177.478,10.797,149.511
C05060=1129.099,335.472,-80.201,-177.476,10.799,149.511
C05061=1129.095,335.685,-80.230,-177.473,10.801,149.511
C05062=1129.091,335.898,-80.259,-177.470,10.803,149.511
C05063=1129.088,336.146,-80.294,-177.467,10.806,149.511
C05064=1129.083,336.393,-80.328,-177.464,10.808,149.510
C05065=1129.080,336.641,-80.362,-177.460,10.811,149.510
C05066=1129.076,336.888,-80.396,-177.457,10.813,149.510
C05067=1129.072,337.136,-80.431,-177.454,10.816,149.510
C05068=1129.068,337.384,-80.464,-177.451,10.818,149.510
C05069=1129.064,337.631,-80.499,-177.448,10.821,149.509
C05070=1129.060,337.879,-80.533,-177.444,10.823,149.509
C05071=1129.056,338.126,-80.567,-177.441,10.826,149.509
C05072=1129.053,338.374,-80.602,-177.438,10.828,149.509
C05073=1129.048,338.622,-80.636,-177.435,10.831,149.509
C05074=1129.045,338.870,-80.670,-177.431,10.833,149.508
C05075=1129.040,339.117,-80.705,-177.428,10.836,149.508
C05076=1129.036,339.364,-80.739,-177.426,10.838,149.508
C05077=1129.032,339.612,-80.774,-177.422,10.840,149.508
C05078=1129.028,339.860,-80.808,-177.419,10.843,149.508
C05079=1129.025,340.107,-80.842,-177.416,10.845,149.507
C05080=1129.020,340.355,-80.877,-177.412,10.848,149.507
C05081=1129.017,340.603,-80.911,-177.410,10.850,149.507
C05082=1129.013,340.849,-80.946,-177.406,10.853,149.507
C05083=1129.009,341.098,-80.981,-177.403,10.855,149.507
C05084=1129.005,341.345,-81.015,-177.400,10.858,149.506
C05085=1129.001,341.593,-81.050,-177.396,10.860,149.506
C05086=1128.996,341.840,-81.084,-177.393,10.863,149.506
C05087=1128.993,342.088,-81.118,-177.390,10.865,149.506
C05088=1128.988,342.335,-81.153,-177.387,10.868,149.506
C05089=1128.985,342.583,-81.188,-177.383,10.870,149.505
C05090=1128.981,342.830,-81.222,-177.380,10.873,149.505
C05091=1128.977,343.078,-81.257,-177.377,10.875,149.505
C05092=1128.972,343.326,-81.292,-177.374,10.878,149.505
C05093=1128.969,343.573,-81.327,-177.371,10.881,149.505
C05094=1128.965,343.821,-81.361,-177.367,10.883,149.505
C05095=1128.961,344.068,-81.396,-177.364,10.885,149.504
C05096=1128.958,344.316,-81.430,-177.361,10.888,149.504
C05097=1128.953,344.563,-81.465,-177.357,10.890,149.504
C05098=1128.949,344.811,-81.500,-177.354,10.893,149.504
C05099=1128.945,345.058,-81.535,-177.351,10.896,149.504
C05100=1128.942,345.306,-81.570,-177.348,10.898,149.503
C05101=1128.938,345.554,-81.604,-177.344,10.900,149.503
C05102=1128.933,345.801,-81.639,-177.342,10.902,149.503
C05103=1128.930,346.049,-81.674,-177.338,10.905,149.503
C05104=1128.925,346.296,-81.709,-177.335,10.907,149.502
C05105=1128.922,346.543,-81.744,-177.332,10.910,149.502
C05106=1128.918,346.791,-81.779,-177.329,10.912,149.502
C05107=1128.914,347.038,-81.814,-177.326,10.915,149.502
C05108=1128.910,347.286,-81.849,-177.322,10.917,149.502
C05109=1128.906,347.534,-81.884,-177.319,10.920,149.501
C05110=1128.902,347.781,-81.919,-177.316,10.922,149.501
C05111=1128.899,347.994,-81.949,-177.313,10.925,149.501
C05112=1128.895,348.207,-81.979,-177.310,10.927,149.501
C05113=1128.893,348.420,-82.009,-177.307,10.928,149.501
C05114=1128.889,348.632,-82.039,-177.304,10.931,149.501
C05115=1128.885,348.846,-82.070,-177.302,10.933,149.500
C05116=1128.882,349.058,-82.099,-177.299,10.936,149.500
C05117=1128.879,349.271,-82.130,-177.296,10.937,149.500
C05118=1128.875,349.484,-82.160,-177.293,10.939,149.500
C05119=1128.872,349.732,-82.194,-177.290,10.942,149.500
C05120=1128.868,349.979,-82.230,-177.286,10.945,149.499
C05121=1128.864,350.227,-82.265,-177.282,10.948,149.499
C05122=1128.860,350.474,-82.300,-177.279,10.950,149.499
C05123=1128.856,350.721,-82.335,-177.275,10.952,149.498
C05124=1128.852,350.969,-82.371,-177.271,10.956,149.498
C05125=1128.848,351.216,-82.405,-177.268,10.958,149.498
C05126=1128.844,351.464,-82.441,-177.264,10.960,149.498
C05127=1128.840,351.711,-82.476,-177.260,10.964,149.497
C05128=1128.837,351.959,-82.512,-177.257,10.966,149.497
C05129=1128.832,352.206,-82.546,-177.254,10.968,149.497
C05130=1128.829,352.454,-82.582,-177.249,10.971,149.497
C05131=1128.825,352.701,-82.617,-177.246,10.974,149.496
C05132=1128.821,352.949,-82.653,-177.243,10.976,149.496
C05133=1128.818,353.196,-82.689,-177.239,10.980,149.496
C05134=1128.813,353.443,-82.724,-177.235,10.982,149.496
C05135=1128.809,353.691,-82.759,-177.232,10.984,149.495
C05136=1128.806,353.939,-82.794,-177.229,10.987,149.495
C05137=1128.802,354.186,-82.830,-177.225,10.990,149.495
C05138=1128.798,354.434,-82.866,-177.221,10.992,149.495
C05139=1128.793,354.681,-82.901,-177.218,10.994,149.494
C05140=1128.790,354.928,-82.937,-177.214,10.997,149.494
C05141=1128.786,355.176,-82.972,-177.210,11.000,149.494
C05142=1128.782,355.423,-83.008,-177.207,11.002,149.493
C05143=1128.779,355.671,-83.043,-177.203,11.005,149.493
C05144=1128.775,355.918,-83.079,-177.200,11.007,149.493
C05145=1128.771,356.165,-83.114,-177.196,11.009,149.493
C05146=1128.766,356.413,-83.150,-177.193,11.012,149.492
C05147=1128.763,356.660,-83.186,-177.189,11.015,149.492
C05148=1128.759,356.908,-83.221,-177.186,11.018,149.492
C05149=1128.755,357.155,-83.257,-177.182,11.020,149.492
C05150=1128.752,357.402,-83.293,-177.179,11.022,149.491
C05151=1128.748,357.650,-83.329,-177.175,11.025,149.491
C05152=1128.743,357.897,-83.364,-177.172,11.027,149.491
C05153=1128.740,358.144,-83.400,-177.168,11.029,149.491
C05154=1128.736,358.392,-83.435,-177.165,11.032,149.490
C05155=1128.732,358.639,-83.471,-177.161,11.035,149.490
C05156=1128.728,358.887,-83.508,-177.157,11.037,149.490
C05157=1128.725,359.134,-83.543,-177.154,11.039,149.490
C05158=1128.721,359.382,-83.579,-177.151,11.042,149.489
C05159=1128.717,359.629,-83.614,-177.148,11.044,149.489
C05160=1128.713,359.876,-83.651,-177.144,11.047,149.489
C05161=1128.710,360.124,-83.687,-177.141,11.049,149.488
C05162=1128.706,360.371,-83.722,-177.137,11.052,149.488
C05163=1128.701,360.619,-83.758,-177.134,11.054,149.488
C05164=1128.698,360.866,-83.795,-177.130,11.056,149.488
C05165=1128.694,361.114,-83.830,-177.127,11.059,149.487
C05166=1128.690,361.361,-83.866,-177.124,11.061,149.487
C05167=1128.686,361.573,-83.897,-177.121,11.063,149.487
C05168=1128.683,361.786,-83.929,-177.118,11.065,149.487
C05169=1128.680,361.999,-83.960,-177.115,11.067,149.486
C05170=1128.677,362.212,-83.990,-177.112,11.069,149.486
C05171=1128.674,362.425,-84.022,-177.109,11.071,149.486
C05172=1128.670,362.636,-84.053,-177.106,11.074,149.486
C05173=1128.667,362.850,-84.083,-177.103,11.076,149.486
C05174=1128.664,363.062,-84.114,-177.101,11.077,149.485
C05175=1128.661,363.309,-84.151,-177.097,11.080,149.485
C05176=1128.656,363.557,-84.187,-177.094,11.082,149.485
C05177=1128.653,363.804,-84.223,-177.090,11.084,149.485
C05178=1128.649,364.051,-84.259,-177.087,11.087,149.484
C05179=1128.645,364.299,-84.296,-177.084,11.089,149.484
C05180=1128.641,364.546,-84.331,-177.080,11.092,149.484
C05181=1128.637,364.793,-84.368,-177.077,11.094,149.484
C05182=1128.634,365.041,-84.404,-177.073,11.096,149.483
C05183=1128.630,365.288,-84.440,-177.070,11.099,149.483
C05184=1128.627,365.536,-84.477,-177.068,11.100,149.483
C05185=1128.622,365.783,-84.513,-177.064,11.103,149.483
C05186=1128.619,366.030,-84.549,-177.061,11.105,149.482
C05187=1128.615,366.277,-84.586,-177.058,11.108,149.482
C05188=1128.611,366.525,-84.622,-177.054,11.110,149.482
C05189=1128.607,366.772,-84.659,-177.051,11.113,149.482
C05190=1128.604,367.019,-84.695,-177.048,11.115,149.482
C05191=1128.599,367.267,-84.731,-177.045,11.117,149.481
C05192=1128.595,367.514,-84.768,-177.041,11.119,149.481
C05193=1128.592,367.761,-84.804,-177.038,11.122,149.481
C05194=1128.588,368.009,-84.840,-177.035,11.124,149.481
C05195=1128.584,368.256,-84.877,-177.031,11.127,149.480
C05196=1128.581,368.504,-84.914,-177.028,11.129,149.480
C05197=1128.577,368.751,-84.951,-177.025,11.131,149.480
C05198=1128.573,368.998,-84.987,-177.022,11.133,149.480
C05199=1128.569,369.245,-85.023,-177.019,11.136,149.479
C05200=1128.565,369.492,-85.059,-177.016,11.138,149.479
C05201=1128.561,369.739,-85.096,-177.012,11.141,149.479
C05202=1128.557,369.987,-85.133,-177.010,11.142,149.479
C05203=1128.555,370.234,-85.170,-177.006,11.145,149.479
C05204=1128.550,370.481,-85.207,-177.003,11.147,149.478
C05205=1128.546,370.729,-85.243,-177.000,11.150,149.478
C05206=1128.543,370.976,-85.280,-176.997,11.151,149.478
C05207=1128.539,371.223,-85.316,-176.994,11.154,149.478
C05208=1128.534,371.471,-85.353,-176.990,11.156,149.478
C05209=1128.531,371.718,-85.390,-176.988,11.159,149.478
C05210=1128.528,371.965,-85.426,-176.985,11.161,149.477
C05211=1128.524,372.212,-85.463,-176.982,11.163,149.477
C05212=1128.519,372.460,-85.500,-176.978,11.166,149.477
C05213=1128.516,372.707,-85.536,-176.975,11.168,149.477
C05214=1128.513,372.954,-85.573,-176.972,11.170,149.476
C05215=1128.509,373.202,-85.610,-176.969,11.173,149.476
C05216=1128.504,373.449,-85.647,-176.966,11.175,149.476
C05217=1128.501,373.695,-85.685,-176.963,11.177,149.476
C05218=1128.498,373.943,-85.721,-176.960,11.180,149.476
C05219=1128.494,374.190,-85.758,-176.957,11.182,149.476
C05220=1128.490,374.437,-85.795,-176.954,11.184,149.475
C05221=1128.486,374.685,-85.832,-176.951,11.187,149.475
C05222=1128.482,374.932,-85.869,-176.948,11.189,149.475
C05223=1128.479,375.145,-85.900,-176.946,11.191,149.475
C05224=1128.476,375.357,-85.932,-176.943,11.193,149.475
C05225=1128.473,375.570,-85.964,-176.941,11.195,149.475
C05226=1128.470,375.782,-85.996,-176.938,11.196,149.474
C05227=1128.466,375.995,-86.028,-176.935,11.199,149.474
C05228=1128.463,376.208,-86.059,-176.932,11.201,149.474
C05229=1128.460,376.420,-86.091,-176.930,11.203,149.474
C05230=1128.456,376.633,-86.123,-176.928,11.205,149.474
C05231=1128.453,376.879,-86.161,-176.925,11.207,149.474
C05232=1128.449,377.126,-86.198,-176.922,11.209,149.474
C05233=1128.445,377.374,-86.235,-176.919,11.212,149.474
C05234=1128.441,377.622,-86.272,-176.916,11.214,149.473
C05235=1128.438,377.868,-86.309,-176.913,11.217,149.473
C05236=1128.434,378.115,-86.346,-176.910,11.219,149.473
C05237=1128.430,378.363,-86.383,-176.908,11.221,149.473
C05238=1128.427,378.609,-86.420,-176.905,11.224,149.473
C05239=1128.422,378.857,-86.457,-176.901,11.226,149.473
C05240=1128.419,379.105,-86.494,-176.899,11.228,149.473
C05241=1128.415,379.351,-86.532,-176.896,11.231,149.473
C05242=1128.411,379.598,-86.569,-176.893,11.233,149.472
C05243=1128.408,379.846,-86.606,-176.891,11.235,149.472
C05244=1128.404,380.093,-86.644,-176.887,11.238,149.472
C05245=1128.400,380.340,-86.681,-176.885,11.240,149.472
C05246=1128.396,380.587,-86.719,-176.882,11.243,149.472
C05247=1128.392,380.834,-86.755,-176.879,11.244,149.472
C05248=1128.389,381.082,-86.793,-176.877,11.247,149.472
C05249=1128.385,381.329,-86.830,-176.874,11.250,149.472
C05250=1128.381,381.575,-86.868,-176.871,11.252,149.472
C05251=1128.378,381.823,-86.905,-176.868,11.255,149.472
C05252=1128.374,382.070,-86.943,-176.866,11.257,149.472
C05253=1128.371,382.318,-86.980,-176.863,11.259,149.472
C05254=1128.367,382.564,-87.017,-176.860,11.262,149.471
C05255=1128.363,382.812,-87.054,-176.857,11.264,149.471
C05256=1128.359,383.059,-87.093,-176.854,11.267,149.471
C05257=1128.355,383.306,-87.130,-176.852,11.269,149.471
C05258=1128.351,383.554,-87.168,-176.850,11.271,149.471
C05259=1128.348,383.800,-87.205,-176.849,11.272,149.471
C05260=1128.344,384.047,-87.242,-176.847,11.275,149.471
C05261=1128.340,384.295,-87.280,-176.846,11.276,149.471
C05262=1128.337,384.541,-87.317,-176.844,11.278,149.472
C05263=1128.333,384.789,-87.355,-176.842,11.280,149.472
C05264=1128.329,385.036,-87.392,-176.841,11.282,149.472
C05265=1128.326,385.284,-87.429,-176.840,11.283,149.472
C05266=1128.321,385.530,-87.468,-176.839,11.285,149.472
C05267=1128.318,385.778,-87.506,-176.837,11.287,149.472
C05268=1128.314,386.024,-87.543,-176.836,11.289,149.472
C05269=1128.310,386.271,-87.580,-176.835,11.291,149.472
C05270=1128.307,386.519,-87.618,-176.833,11.293,149.473
C05271=1128.303,386.765,-87.656,-176.832,11.295,149.473
C05272=1128.300,387.013,-87.693,-176.831,11.297,149.473
C05273=1128.295,387.260,-87.731,-176.829,11.299,149.473
C05274=1128.292,387.507,-87.769,-176.828,11.300,149.473
C05275=1128.288,387.755,-87.806,-176.827,11.302,149.473
C05276=1128.285,388.002,-87.844,-176.825,11.305,149.474
C05277=1128.281,388.248,-87.881,-176.824,11.307,149.474
C05278=1128.278,388.496,-87.919,-176.823,11.309,149.474
C05279=1128.274,388.708,-87.952,-176.821,11.311,149.474
C05280=1128.271,388.920,-87.984,-176.820,11.313,149.475
C05281=1128.268,389.133,-88.016,-176.820,11.315,149.475
C05282=1128.264,389.345,-88.048,-176.818,11.316,149.475
C05283=1128.261,389.558,-88.081,-176.817,11.318,149.475
C05284=1128.258,389.771,-88.114,-176.817,11.320,149.475
C05285=1128.255,389.983,-88.146,-176.815,11.322,149.476
C05286=1128.252,390.195,-88.178,-176.814,11.324,149.476
C05287=1128.249,390.442,-88.216,-176.814,11.325,149.476
C05288=1128.245,390.689,-88.254,-176.812,11.328,149.476
C05289=1128.241,390.937,-88.292,-176.811,11.330,149.477
C05290=1128.237,391.184,-88.329,-176.810,11.333,149.477
C05291=1128.234,391.431,-88.367,-176.809,11.335,149.477
C05292=1128.230,391.678,-88.405,-176.808,11.337,149.478
C05293=1128.226,391.925,-88.443,-176.807,11.340,149.478
C05294=1128.222,392.172,-88.481,-176.807,11.342,149.478
C05295=1128.219,392.419,-88.519,-176.805,11.344,149.479
C05296=1128.215,392.666,-88.556,-176.804,11.346,149.479
C05297=1128.212,392.913,-88.594,-176.803,11.349,149.480
C05298=1128.207,393.160,-88.632,-176.802,11.351,149.480
C05299=1128.204,393.408,-88.670,-176.801,11.354,149.480
C05300=1128.200,393.654,-88.707,-176.801,11.357,149.481
C05301=1128.196,393.902,-88.746,-176.800,11.358,149.481
C05302=1128.192,394.148,-88.783,-176.799,11.361,149.482
C05303=1128.189,394.396,-88.821,-176.798,11.364,149.482
C05304=1128.186,394.643,-88.859,-176.797,11.367,149.483
C05305=1128.181,394.890,-88.897,-176.797,11.369,149.483
C05306=1128.178,395.137,-88.935,-176.796,11.372,149.484
C05307=1128.175,395.384,-88.973,-176.795,11.374,149.484
C05308=1128.171,395.631,-89.011,-176.794,11.377,149.485
C05309=1128.167,395.878,-89.049,-176.793,11.380,149.485
C05310=1128.164,396.125,-89.087,-176.793,11.382,149.485
C05311=1128.159,396.372,-89.125,-176.791,11.385,149.486
C05312=1128.156,396.619,-89.163,-176.791,11.388,149.486
C05313=1128.153,396.866,-89.201,-176.790,11.391,149.487
C05314=1128.148,397.113,-89.239,-176.790,11.393,149.488
C05315=1128.145,397.361,-89.277,-176.789,11.396,149.488
C05316=1128.141,397.607,-89.315,-176.789,11.399,149.489
C05317=1128.137,397.855,-89.353,-176.788,11.402,149.489
C05318=1128.133,398.101,-89.391,-176.787,11.405,149.490
C05319=1128.130,398.349,-89.429,-176.787,11.408,149.491
C05320=1128.126,398.596,-89.467,-176.786,11.411,149.491
C05321=1128.123,398.843,-89.505,-176.786,11.413,149.492
C05322=1128.119,399.090,-89.543,-176.785,11.417,149.492
C05323=1128.115,399.337,-89.581,-176.784,11.420,149.493
C05324=1128.112,399.584,-89.619,-176.784,11.422,149.494
C05325=1128.108,399.832,-89.657,-176.784,11.426,149.494
C05326=1128.104,400.078,-89.695,-176.783,11.429,149.495
C05327=1128.101,400.326,-89.733,-176.783,11.432,149.496
C05328=1128.096,400.572,-89.771,-176.782,11.435,149.497
C05329=1128.093,400.819,-89.810,-176.781,11.438,149.497
C05330=1128.089,401.067,-89.848,-176.782,11.441,149.498
C05331=1128.086,401.313,-89.886,-176.781,11.445,149.499
C05332=1128.082,401.561,-89.924,-176.780,11.448,149.499
C05333=1128.078,401.807,-89.962,-176.781,11.451,149.500
C05334=1128.075,402.055,-90.000,-176.780,11.454,149.501
C05335=1128.071,402.267,-90.033,-176.780,11.457,149.502
C05336=1128.069,402.479,-90.066,-176.779,11.460,149.502
C05337=1128.065,402.692,-90.099,-176.779,11.463,149.503
C05338=1128.062,402.904,-90.131,-176.779,11.466,149.504
C05339=1128.059,403.116,-90.165,-176.779,11.469,149.504
C05340=1128.056,403.329,-90.198,-176.779,11.472,149.505
C05341=1128.053,403.541,-90.230,-176.778,11.475,149.506
C05342=1128.050,403.753,-90.262,-176.778,11.478,149.507
C05343=1128.046,404.000,-90.301,-176.778,11.481,149.507
C05344=1128.042,404.247,-90.339,-176.778,11.485,149.508
C05345=1128.038,404.494,-90.378,-176.778,11.488,149.509
C05346=1128.035,404.742,-90.416,-176.778,11.492,149.510
C05347=1128.031,404.988,-90.454,-176.778,11.496,149.511
C05348=1128.028,405.235,-90.492,-176.777,11.499,149.512
C05349=1128.024,405.483,-90.531,-176.777,11.503,149.513
C05350=1128.020,405.729,-90.568,-176.777,11.507,149.514
C05351=1128.017,405.976,-90.607,-176.778,11.510,149.515
C05352=1128.013,406.224,-90.646,-176.777,11.514,149.516
C05353=1128.009,406.470,-90.683,-176.778,11.518,149.517
C05354=1128.005,406.718,-90.722,-176.778,11.522,149.518
C05355=1128.002,406.964,-90.760,-176.777,11.525,149.519
C05356=1127.998,407.211,-90.799,-176.777,11.529,149.520
C05357=1127.995,407.459,-90.837,-176.777,11.533,149.521
C05358=1127.991,407.705,-90.876,-176.778,11.537,149.522
C05359=1127.987,407.952,-90.913,-176.778,11.541,149.523
C05360=1127.983,408.200,-90.952,-176.778,11.545,149.524
C05361=1127.981,408.446,-90.991,-176.778,11.550,149.525
C05362=1127.976,408.693,-91.029,-176.778,11.554,149.526
C05363=1127.973,408.940,-91.067,-176.778,11.558,149.527
C05364=1127.969,409.187,-91.106,-176.779,11.562,149.529
C05365=1127.966,409.435,-91.144,-176.779,11.566,149.530
C05366=1127.961,409.682,-91.182,-176.779,11.570,149.531
C05367=1127.958,409.929,-91.221,-176.779,11.574,149.532
C05368=1127.955,410.176,-91.259,-176.780,11.579,149.533
C05369=1127.950,410.423,-91.297,-176.780,11.583,149.535
C05370=1127.947,410.669,-91.336,-176.780,11.587,149.536
C05371=1127.943,410.917,-91.375,-176.781,11.591,149.537
C05372=1127.940,411.163,-91.412,-176.781,11.596,149.538
C05373=1127.936,411.410,-91.451,-176.782,11.600,149.539
C05374=1127.933,411.658,-91.489,-176.782,11.604,149.541
C05375=1127.929,411.905,-91.529,-176.783,11.609,149.542
C05376=1127.925,412.152,-91.567,-176.783,11.613,149.543
C05377=1127.922,412.398,-91.605,-176.784,11.617,149.544
C05378=1127.918,412.646,-91.644,-176.784,11.623,149.546
C05379=1127.915,412.893,-91.682,-176.785,11.627,149.547
C05380=1127.910,413.139,-91.721,-176.785,11.632,149.548
C05381=1127.906,413.387,-91.759,-176.786,11.636,149.550
C05382=1127.904,413.634,-91.798,-176.787,11.641,149.551
C05383=1127.900,413.881,-91.836,-176.787,11.646,149.553
C05384=1127.896,414.127,-91.875,-176.787,11.651,149.554
C05385=1127.894,414.375,-91.913,-176.788,11.655,149.555
C05386=1127.891,414.622,-91.952,-176.789,11.660,149.557
C05387=1127.889,414.869,-91.990,-176.790,11.665,149.558
C05388=1127.888,415.115,-92.028,-176.790,11.670,149.560
C05389=1127.888,415.363,-92.066,-176.791,11.675,149.561
C05390=1127.888,415.610,-92.104,-176.792,11.680,149.563
C05391=1127.889,415.822,-92.137,-176.793,11.684,149.564
C05392=1127.889,416.034,-92.170,-176.793,11.689,149.565
C05393=1127.891,416.246,-92.202,-176.794,11.692,149.567
C05394=1127.892,416.459,-92.234,-176.795,11.697,149.568
C05395=1127.895,416.670,-92.267,-176.796,11.701,149.569
C05396=1127.897,416.883,-92.300,-176.796,11.706,149.571
C05397=1127.901,417.094,-92.331,-176.798,11.710,149.572
C05398=1127.904,417.307,-92.364,-176.799,11.714,149.573
C05399=1127.485,417.307,-92.426,-176.791,11.719,149.573
C05400=1127.482,417.094,-92.394,-176.790,11.715,149.571
C05401=1127.478,416.882,-92.362,-176.789,11.710,149.570
C05402=1127.476,416.670,-92.329,-176.789,11.706,149.569
C05403=1127.473,416.459,-92.297,-176.788,11.701,149.567
C05404=1127.472,416.246,-92.265,-176.787,11.697,149.566
C05405=1127.470,416.034,-92.232,-176.786,11.693,149.565
C05406=1127.469,415.821,-92.200,-176.785,11.689,149.563
C05407=1127.468,415.610,-92.167,-176.785,11.684,149.562
C05408=1127.469,415.362,-92.129,-176.784,11.679,149.561
C05409=1127.469,415.115,-92.091,-176.784,11.674,149.559
C05410=1127.470,414.869,-92.053,-176.783,11.669,149.558
C05411=1127.472,414.622,-92.014,-176.782,11.665,149.556
C05412=1127.474,414.374,-91.975,-176.782,11.659,149.555
C05413=1127.477,414.128,-91.937,-176.781,11.654,149.553
C05414=1127.480,413.880,-91.899,-176.780,11.650,149.552
C05415=1127.484,413.633,-91.860,-176.780,11.645,149.551
C05416=1127.487,413.386,-91.822,-176.779,11.640,149.549
C05417=1127.491,413.140,-91.783,-176.779,11.635,149.548
C05418=1127.495,412.892,-91.744,-176.778,11.631,149.547
C05419=1127.498,412.645,-91.706,-176.777,11.626,149.545
C05420=1127.502,412.399,-91.667,-176.778,11.621,149.544
C05421=1127.506,412.152,-91.629,-176.777,11.617,149.543
C05422=1127.509,411.905,-91.590,-176.777,11.613,149.541
C05423=1127.513,411.657,-91.552,-176.776,11.608,149.540
C05424=1127.517,411.411,-91.513,-176.775,11.604,149.539
C05425=1127.521,411.163,-91.475,-176.776,11.599,149.538
C05426=1127.523,410.917,-91.436,-176.775,11.595,149.536
C05427=1127.527,410.669,-91.398,-176.775,11.590,149.535
C05428=1127.532,410.422,-91.360,-176.775,11.586,149.534
C05429=1127.535,410.176,-91.321,-176.774,11.582,149.533
C05430=1127.539,409.928,-91.282,-176.774,11.578,149.532
C05431=1127.542,409.682,-91.244,-176.774,11.573,149.530
C05432=1127.546,409.435,-91.205,-176.773,11.569,149.529
C05433=1127.549,409.187,-91.168,-176.773,11.565,149.528
C05434=1127.553,408.940,-91.128,-176.773,11.561,149.527
C05435=1127.557,408.694,-91.091,-176.773,11.557,149.526
C05436=1127.561,408.446,-91.052,-176.772,11.553,149.525
C05437=1127.564,408.200,-91.014,-176.773,11.548,149.524
C05438=1127.568,407.953,-90.975,-176.773,11.544,149.523
C05439=1127.571,407.705,-90.937,-176.773,11.540,149.521
C05440=1127.575,407.458,-90.898,-176.773,11.536,149.520
C05441=1127.579,407.212,-90.861,-176.772,11.533,149.519
C05442=1127.583,406.964,-90.822,-176.772,11.529,149.518
C05443=1127.585,406.718,-90.783,-176.772,11.525,149.517
C05444=1127.589,406.470,-90.745,-176.772,11.521,149.516
C05445=1127.593,406.223,-90.707,-176.772,11.517,149.515
